// TwinCAT 3 PLC project PLC1
// ProgramVersion: 3.1.4024.0
// libraries:
//   Tc2_EtherCAT, * (Beckhoff Automation GmbH)
//   Tc2_MC2, * (Beckhoff Automation GmbH)
//   Tc2_Standard, * (Beckhoff Automation GmbH)
//   Tc2_System, * (Beckhoff Automation GmbH)
//   Tc3_Module, * (Beckhoff Automation GmbH)
// project tree:
//   DUTs/Dosing Pumps/ E_AccessType.TcDUT, E_DosingPump.TcDUT, E_ModbusDataType.TcDUT, ST_EmcoPumpModbusData.TcDUT, ST_ModbusRegister.TcDUT
//   DUTs/ E_ConveyorMoveType.TcDUT, E_DeviceState.TcDUT, E_LinActuatorMoveType.TcDUT, E_MoveState.TcDUT, E_TrayExchangeState.TcDUT, ST_INPUTS_LinAct.TcDUT, ST_INPUTS_POP.TcDUT, ST_INPUTS_LFT.TcDUT, ST_INPUTS_SequenceManager_POP.TcDUT, ST_INPUTS_StaticConv.TcDUT, ST_INPUTS_TrayCentre.TcDUT
//   DUTs/GVL/Inputs/Dosing Machine/Children/ ST_INPUTS_DosingMachine_Sump.TcDUT, ST_INPUTS_DosingMachine_Water.TcDUT
//   DUTs/GVL/Inputs/Dosing Machine/ ST_INPUTS_DosingMachine.TcDUT
//   DUTs/GVL/Inputs/RND_DM/Children/ ST_INPUTS_RND_DosingMachine_Sump.TcDUT, ST_INPUTS_RND_DosingMachine_Water.TcDUT
//   DUTs/GVL/Inputs/RND_DM/ ST_INPUTS_RND_DosingMachine.TcDUT
//   DUTs/GVL/Inputs/RND_SC/ ST_INPUTS_RND_LevelWaterControl.TcDUT, ST_INPUTS_RND_StackControl.TcDUT
//   DUTs/GVL/Inputs/RND_WTR/ ST_INPUTS_WaterTreatment_RND.TcDUT
//   DUTs/GVL/Inputs/Universal/ ST_INPUTS_BagFilters.TcDUT, ST_INPUTS_Calibration.TcDUT, ST_INPUTS_ControlLoop_BangBang.TcDUT, ST_INPUTS_ControlLoop_BangBangAnalog.TcDUT, ST_INPUTS_DosingPump.TcDUT, ST_INPUTS_Dosing_ControlLoop.TcDUT, ST_INPUTS_DrumFilter.TcDUT, ST_INPUTS_PumpDOL.TcDUT, ST_INPUTS_PumpVSD.TcDUT, ST_INPUTS_RND_HVAC_Indoor_Unit.TcDUT, ST_INPUTS_SequenceManager_DM.TcDUT, ST_INPUTS_SequenceManager_RND_DM.TcDUT, ST_INPUTS_Strainer.TcDUT, ST_INPUTS_Unit_OxyInjector.TcDUT, ST_INPUTS_Unit_OzoneGenerator.TcDUT, ST_INPUTS_Unit_RO_EDI.TcDUT, ST_INPUTS_Unit_UltraSonCleaner.TcDUT, ST_INPUTS_Unit_UVFilter.TcDUT, ST_INPUTS_ValveOnOFF.TcDUT
//   DUTs/GVL/Inputs/Water Treatment/ ST_INPUTS_WaterTreatment.TcDUT, ST_INPUTS_WaterTreatment_Water.TcDUT
//   DUTs/Machines/ E_MachineState.TcDUT, ST_DMComponents.TcDUT, ST_POPComponents.TcDUT, ST_LFTComponents.TcDUT, ST_RNDDMComponents.TcDUT, ST_RNDWTRComponents.TcDUT, ST_WTRComponents.TcDUT
//   DUTs/Universal/ E_AlarmPriority.TcDUT, E_DeviceMode.TcDUT, E_InterlockType.TcDUT, E_Job_Status.TcDUT, E_POP_Type.TcDUT, E_SensorType.TcDUT, E_SequenceList_DM.TcDUT, E_SequenceList_POP.TcDUT, E_SequenceList_RND_DM.TcDUT, E_SequenceList_WTR.TcDUT, E_SequenceState.TcDUT, ST_Alarm.TcDUT, ST_Crop.TcDUT, ST_CropJob.TcDUT, ST_HandShake_TrayMovement.TcDUT, ST_HVAC.TcDUT, ST_Interlock.TcDUT, ST_Modbus_ReadRequest.TcDUT, ST_Modbus_WriteRequest.TcDUT, ST_OEE.TcDUT, ST_PlantConfig.TcDUT, ST_SequenceStep.TcDUT, ST_Tray.TcDUT, ST_TrayExchangeHandshake.TcDUT, ST_Tray_1.TcDUT, ST_Tray_2.TcDUT
//   GVLs/ GVL.TcGVL, Inputs.TcGVL, IO_MAPPING.TcGVL, Safety.TcGVL
//   / MAIN.TcPOU, PlcTask.TcTTO
//   POUs/00 Interfaces/ FB_BaseDevice.TcPOU, FB_BaseMachine.TcPOU, FB_BaseMachine_1.TcPOU, FB_BaseSensor.TcPOU, FB_HandShake_TrayMovement.TcPOU, I_Device.TcIO, I_Machine.TcIO, I_PumpDosing.TcIO, I_PumpVSD.TcIO, I_Sensor.TcIO, I_Sequence.TcIO, I_ValveActuated.TcIO
//   POUs/01 Actuators/Dosing Machine/ FB_AutoClean_Filter_Bollfilter.TcPOU, FB_DosingPumpAgrowtek_R2.TcPOU, FB_DosingPumpAgrowtek_R2_1.TcPOU, FB_DosingPumpAgrowtek_R2_Batch.TcPOU, FB_DosingPumpPRISMA.TcPOU, FB_DrumFilter_Faivre120.TcPOU, FB_DrumFilter_Faivre60.TcPOU, FB_GasMonitoringPanel_CDA4022.TcPOU, FB_GasMonitoringPanel_CDA4022_R2.TcPOU, FB_HVAC_RND_Indoor_Unit.TcPOU, FB_HVAC_RND_ModbusApadtor.TcPOU, FB_LevelWaterControl.TcPOU, FB_OxygenInjector.TcPOU, FB_OxygenInjector_1.TcPOU, FB_OzoneGenerator.TcPOU, FB_PumpDOL_Onga413.TcPOU, FB_PumpDOL_Onga413_RND.TcPOU, FB_PumpVSD_DanfossFC202.TcPOU, FB_PumpVSD_GrundfosCUE.TcPOU, FB_UltraSonicCleaner.TcPOU, FB_Unit_RO_PW30_1.TcPOU, FB_Unit_RO_RND.TcPOU, FB_UVFilter_Pentair_EU40.TcPOU, FB_UVFilter_UltraAqua_MR4_220PP.TcPOU
//   POUs/01 Actuators/ FB_Valve_ONOFF_woMonitoring.TcPOU, FB_Valve_ONOFF_woMonitoring_1.TcPOU
//   POUs/01 Actuators/supersceded/ FB_DosingPumpAgrowtek.TcPOU
//   POUs/02 Sensors/Dosing Machine/ FB_Sensor_AtlasDO.TcPOU, FB_Sensor_AtlasEC.TcPOU, FB_Sensor_AtlasORP.TcPOU, FB_Sensor_AtlasPH.TcPOU, FB_Sensor_AtlasTEMP.TcPOU, FB_Sensor_GrowMedium_EC.TcPOU, FB_Sensor_GrowMedium_MOISTURE.TcPOU, FB_Sensor_GrowMedium_PH.TcPOU, FB_Sensor_IFM_PG2453.TcPOU, FB_Sensor_OceanControlsPressureTx_BVS006NA.TcPOU, FB_Sensor_SICKLevelSwitch_GRF18S.TcPOU
//   POUs/02 Sensors/ FB_DualRedundantSensor.TcPOU, FB_Sensor_4_20mA_Generic.TcPOU, FB_Sensor_VaisalaGMW90.TcPOU, FB_Sensor_VaisalaGMW90_R2.TcPOU, FB_Sensor_VaisalaGMW90_R2_1.TcPOU
//   POUs/03 Physical Entities/ FB_BagFilter.TcPOU, FB_Tank.TcPOU
//   POUs/04 Control Loops/Dosing Machine/ FB_BangBangControl.TcPOU, FB_BangBangControl_Analog.TcPOU, FB_BatchController_Dosing.TcPOU, FB_ControlLoop_DissOx.TcPOU, FB_ControlLoop_Dosing.TcPOU, FB_ControlLoop_HVAC.TcPOU, FB_ControlLoop_HVAC_1.TcPOU, FB_ControlLoop_MainPumpPressure.TcPOU, FB_ControlLoop_pH.TcPOU, FB_ControlLoop_PID.TcPOU, FB_ControlLoop_PID_HVAC.TcPOU, FB_ControlLoop_TankLevel.TcPOU
//   POUs/04 Control Loops/_ss/ FB_ControlLoop_Dosing_1.TcPOU
//   POUs/05 Sequences/Dosing Machine/ FB_SequenceDM_Calibrate.TcPOU, FB_SequenceDM_Drain.TcPOU, FB_SequenceDM_Fill.TcPOU, FB_SequenceDM_Main.TcPOU
//   POUs/05 Sequences/ FB_SequenceBase.TcPOU, FB_SequenceManager.TcPOU, FB_SequenceManager_1.TcPOU, FB_SequenceManager_ss.TcPOU
//   POUs/05 Sequences/POP/ FB_SequenceCONVEY_EXTEND.TcPOU, FB_SequenceCONVEY_RETRACT.TcPOU, FB_SequenceEXTEND_CONVEY.TcPOU, FB_SequenceGET_READY_EXTEND.TcPOU, FB_SequenceGET_READY_RETRACT.TcPOU, FB_SequenceRETRACT_CONVEY.TcPOU
//   POUs/05 Sequences/LFT/ FB_SequenceMOVE.TcPOU
//   POUs/05 Sequences/RnD Machines/ FB_SequenceRNDWTR_Main.TcPOU, FB_SequenceRND_Calibrate.TcPOU, FB_SequenceRND_Drain.TcPOU, FB_SequenceRND_Fill.TcPOU, FB_SequenceRND_FirstDose.TcPOU, FB_SequenceRND_Flush.TcPOU, FB_SequenceRND_Main.TcPOU
//   POUs/05 Sequences/Water Treatment/ FB_SequenceWTR_Calibrate.TcPOU, FB_SequenceWTR_Main.TcPOU
//   POUs/06 Machines/ FB_Machine_LFT.TcPOU
//   POUs/06 Machines/Others/ FB_Machine_DosingMachine.TcPOU, FB_Machine_RND_DosingMachine_R2.TcPOU, FB_Machine_RND_DosingMachine_R2_1.TcPOU, FB_Machine_WaterTreatment.TcPOU, FB_Machine_WaterTreatment_RND.TcPOU, FB_Stack_Controller.TcPOU, FB_Stack_Controller_RND.TcPOU
//   POUs/06 Machines/_ss/ FB_Machine_DosingMachine_TEST2.TcPOU, FB_Machine_RND_DosingMachine.TcPOU
//   POUs/07 Systems/RND/ FB_System_RND_GasMonitoring.TcPOU, FB_System_RND_GasMonitoring_R2.TcPOU, FB_System_RND_HVAC.TcPOU
//   POUs/97 Signal Conditioning/ FB_SigCond_MovingAverage.TcPOU
//   POUs/99 Utilities/ FB_HealthMonitoring.TcPOU, FB_InterlockManager.TcPOU, FB_ModbusManager.TcPOU, FB_ModbusMaster_R2.TcPOU, FB_RS485_CardRead.TcPOU, FB_RS485_CardWrite.TcPOU, FB_SensorVirtual_Vaisala.TcPOU, FB_TimeStampProvider.TcPOU
//   POUs/99 Utilities/_ss/ FB_ModbusManager_1.TcPOU, FB_ModbusMaster.TcPOU, FB_ModbusMaster_R2_1.TcPOU
//   POUs/LFT/ E_AxisNumberCoE.TcDUT, E_CoEService.TcDUT, E_ConfigurationStateCoE.TcDUT, E_MovidriveB_OpMode.TcDUT, FB_AutoGreaser.TcPOU, FB_Lift.TcPOU, FB_LiftArm.TcPOU, FB_ParameterCoE_ReadWrite_GenC.TcPOU, FB_SEW_MovidriveB.TcPOU, ST_StackDestination.TcDUT
//   POUs/POP/ FB_ActuatorLinear.TcPOU, FB_AutoSwitch.TcPOU, FB_BaseMotor.TcPOU, FB_LinearActuator_Elec.TcPOU, FB_LinearActuator_Pneumatic.TcPOU, FB_Sensor_OMRON_E3AS.TcPOU, FB_StaticConveyor.TcPOU
// real-time tasks:
//   TASK PlcTask: cycle T#10ms, priority 20, ADS port 350
// I/O:
//   DEVICE CONTROL_BOX, AmsNetId 192.168.1.31.2.1
//     Term 1 (EK1200) [EK1200-5000 EtherCAT Power supply (2A E-Bus)]
//       Term 8 (EL6070) [EL6070 1Ch. Licensing-Terminal]
//       Term 9 (EL6910) [EL6910, TwinSAFE PLC]
//       Term 10 (EL1904) [EL1904, 4 Ch. Safety Input 24V, TwinSAFE]
//         modules: Module 1 (FSOES)
//       Term 11 (EL1008) [EL1008 8Ch. Dig. Input 24V, 3ms]
//       Term 12 (EL1904) [EL1904, 4 Ch. Safety Input 24V, TwinSAFE]
//         modules: Module 1 (FSOES)
//       Term 13 (EL1904) [EL1904, 4 Ch. Safety Input 24V, TwinSAFE]
//         modules: Module 1 (FSOES)
//       Term 14 (EL2008) [EL2008 8Ch. Dig. Output 24V, 0.5A]
//       Term 15 (EL2904) [EL2904, 4 Ch. Safety Output 24V, 0.5A, TwinSAFE]
//         modules: Module 1 (FSOES), Module 2 (DO)
//       Term 10 (EL9011) [EL9011 End Terminal]
//   DEVICE Device 4 (EtherCAT), AmsNetId 192.168.1.31.5.1
//     Box 1 (EP1008-0002) [EP1008-0002 8 Ch. Dig. Input 24V, 3ms, M12]
//     Box 2 (EP2308-0002) [EP2308-0002 4 CH. Dig. In, 3ms, 4 Ch. Dig. Out 24V, 0,5A, M12]
//     Drive 3 (MOVIDRIVE+DFE24) [MOVIDRIVE+DFE24]
// variable links:
//   CONTROL_BOX <-> CONTROL_BOX/Term 1 (EK1200)/Term 12 (EL1904)
//     Term 1 (EK1200)/Term 9 (EL6910)/ConnectionOutputs/Message_3 RxPDO <-> Module 1 (FSOES)/TxPDO/FSOE
//   CONTROL_BOX <-> CONTROL_BOX/Term 1 (EK1200)/Term 9 (EL6910)
//     Term 1 (EK1200)/Term 10 (EL1904)/Module 1 (FSOES)/RxPDO/FSOE <-> ConnectionInputs/Message_2 TxPDO
//     Term 1 (EK1200)/Term 12 (EL1904)/Module 1 (FSOES)/RxPDO/FSOE <-> ConnectionInputs/Message_3 TxPDO
//     Term 1 (EK1200)/Term 13 (EL1904)/Module 1 (FSOES)/RxPDO/FSOE <-> ConnectionInputs/Message_4 TxPDO
//     Term 1 (EK1200)/Term 15 (EL2904)/Module 1 (FSOES)/RxPDO/FSOE <-> ConnectionInputs/Message_5 TxPDO
//     Term 1 (EK1200)/Term 10 (EL1904)/Module 1 (FSOES)/TxPDO/FSOE <-> ConnectionOutputs/Message_2 RxPDO
//     Term 1 (EK1200)/Term 13 (EL1904)/Module 1 (FSOES)/TxPDO/FSOE <-> ConnectionOutputs/Message_4 RxPDO
//     Term 1 (EK1200)/Term 15 (EL2904)/Module 1 (FSOES)/TxPDO/FSOE <-> ConnectionOutputs/Message_5 RxPDO
//   PLC1/PLC1 Instance <-> CONTROL_BOX/Term 1 (EK1200)/Term 11 (EL1008)
//     PlcTask Inputs/MAIN.fbMachine_Lift.fbSensor_PressSwitch.bRawInput <-> Channel 3/Input
//   PLC1/PLC1 Instance <-> CONTROL_BOX/Term 1 (EK1200)/Term 14 (EL2008)
//     PlcTask Outputs/MAIN.fbMachine_Lift.bLOCK_CTRL <-> Channel 3/Output
//     PlcTask Outputs/MAIN.fbMachine_Lift.bPWR_CTRL <-> Channel 1/Output
//   PLC1/PLC1 Instance <-> CONTROL_BOX/Term 1 (EK1200)/Term 9 (EL6910)
//     PlcTask Outputs/Safety.bSafetyErrorAcknowledge <-> StandardOutputs/Standard In Var 1
//     PlcTask Outputs/Safety.bSafety_Run_Stop <-> StandardOutputs/Standard In Var 7
//   PLC1/PLC1 Instance <-> Device 4 (EtherCAT)/Box 1 (EP1008-0002)
//     PlcTask Inputs/MAIN.fbMachine_Lift.fbSensor_LiftBrake_Left.bRawInput <-> Channel 8/Input
//     PlcTask Inputs/MAIN.fbMachine_Lift.fbSensor_LiftBrake_Right.bRawInput <-> Channel 7/Input
//     PlcTask Inputs/MAIN.fbMachine_Lift.fbSensor_Lift_Bottom.bRawInput <-> Channel 3/Input
//     PlcTask Inputs/MAIN.fbMachine_Lift.fbSensor_Lift_Home.bRawInput <-> Channel 1/Input
//     PlcTask Inputs/MAIN.fbMachine_Lift.fbSensor_Lift_Top.bRawInput <-> Channel 2/Input
//   PLC1/PLC1 Instance <-> Device 4 (EtherCAT)/Box 2 (EP2308-0002)
//     PlcTask Outputs/MAIN.bGreaser <-> Channel 5/Output
//     PlcTask Outputs/MAIN.bGreaser2 <-> Channel 6/Output
//     PlcTask Outputs/MAIN.fbMachine_Lift.fbValve_Brake.bValveOutput <-> Channel 8/Output
//     PlcTask Outputs/MAIN.fbMachine_Lift.fbValve_Vacuum.bValveOutput <-> Channel 7/Output

CONFIGURATION PLC1
    RESOURCE PLC ON TwinCAT3
        TASK PlcTask(INTERVAL := T#10ms, PRIORITY := 20);
        PROGRAM MAIN WITH PlcTask : MAIN;
    END_RESOURCE
END_CONFIGURATION

// ---- DUTs/Dosing Pumps/E_AccessType.TcDUT
{attribute 'qualified_only'}
{attribute 'strict'}
TYPE E_AccessType :
(
	READ,
	WRITE,
	READWRITE
);
END_TYPE

// ---- DUTs/Dosing Pumps/E_DosingPump.TcDUT
{attribute 'qualified_only'}
{attribute 'strict'}
TYPE E_DosingPump :
(
	PH_UP := 0,
	PH_DOWN := 1,
	NUTRIENT_A := 2,
	NUTRIENT_B := 3,
	NUTRIENT_C := 4
);
END_TYPE

// ---- DUTs/Dosing Pumps/E_ModbusDataType.TcDUT
{attribute 'qualified_only'}
{attribute 'strict'}
TYPE E_ModbusDataType :
(
	uint16,
	uint32,
	uint64
);
END_TYPE

// ---- DUTs/Dosing Pumps/ST_EmcoPumpModbusData.TcDUT
TYPE ST_EmcoPumpModbusData :
STRUCT
	ALARM_Level_Alarm:  UINT;
	ALARM_Pump_Status_When_Level_Alarm_Occurs:  UINT;
	ALARM_Stand_By:  UINT;
	ALARM_Overflow:  UINT;
	ALARM_Temperature:  UINT;
	ALARM_No_Input:  UINT;
	ALARM_Overpressure:  UINT;
	DOSAGE_Dosage_Schedule:  UDINT;
	DOSAGE_Frequency:  UDINT;
	SETTINGS_Level_Alarm:  UINT;
	SETTINGS_Level_Alarm_Contact:  UINT;
	SETTINGS_Reserve_Level_Alarm:  UDINT;
	SETTINGS_Unit:  UINT;
	MODE_Working_Mode:  UINT;
	SETTINGS_Water_Meter_Input_Unit_Of_Measure:  UINT;
	SETTINGS_Water_Meter_Input_Value:  UINT;
	STATISTICS_Partial_Statistics_Dosato:  ULINT;
	STATISTICS_Partial_Statistics_Counter:  ULINT;
	STATISTICS_Partial_Statistics_Dosato_In_The_Last_24H:  ULINT;
	STATISTICS_Partial_Statistics_Counter_In_The_Last_24H:  ULINT;
	STATISTICS_Partial_Statistics_Reset_The_Last_Time_Hrs:  UINT;
	STATISTICS_Partial_Statistics_Reset_The_Last_Time_Mins:  UINT;
	STATISTICS_Partial_Statistics_Reset_The_Last_Time_Seconds:  UINT;
	STATISTICS_Partial_Statistics_Date_Last_Reset_Day:  UINT;
	STATISTICS_Partial_Statistics_Date_Last_Reset_Month:  UINT;
	STATISTICS_Partial_Statistics_Date_Last_Reset_Year:  UINT;
	STATISTICS_Statistics_Total_Total_Dosage:  ULINT;
	STATISTICS_Statistics_Total_Counter:  ULINT;
	MODE_ON_OFF:  UINT;
	SETTINGS_Timeout_Val:  UINT;
	SETTINGS_Overflow_Val:  UINT;
	SETTINGS_Delay:  UINT;
	MODE_Constant_Mode:  UDINT;
	MODE_Mode_Ppm:  UDINT;
	MODE_Mode_Ppm_Concentration:  UINT;
	MODE_Mode_Perc:  UDINT;
	MODE_Mode_Perc_Concentration:  UINT;
	MODE_Mode_Mlq:  UDINT;
	MODE_Mode_Mlq_Concentration:  UINT;
	MODE_Method_Volt_Volt_High_Value:  UINT;
	MODE_Method_Volt_Volt_Low_Value:  UINT;
	MODE_Method_Volt_High_Dose:  UDINT;
	MODE_Mode_Volt_Low_Dose:  UDINT;
	MODE_Method_Ma_Ma_High_Value:  UINT;
	MODE_Method_Ma_Ma_Low_Value:  UINT;
	MODE_Method_Ma_High_Dosage:  UDINT;
	MODE_Method_Ma_Low_Dosage:  UDINT;
	MODE_Pulse_Mode_Pulse_High_Value:  UINT;
	MODE_Pulse_Mode_Pulse_Low_Value:  UINT;
	MODE_Pulse_Mode_High_Dose:  UDINT;
	MODE_Pulse_Low_Dose:  UDINT;
	MODE_Method_Pause_Minutes_Work_Work:  UINT;
	MODE_Method_Pause_Minutes_Of_Work_Pause:  UINT;
	MODE_Method_Pause_Quantity_Work_To_Dose:  UDINT;
	SETTINGS_Flow:  UDINT;
	SETTINGS_Slow_Mode:  UINT;
	SETTINGS_Alarm_Output:  UINT;
	SETTINGS_Alarm_Output_Contact_0_No_1_Nc:  UINT;
	SETTINGS_Alarm_Output_Alert_Level:  UINT;
	SETTINGS_Alarm_Out_Standby:  UINT;
	SETTINGS_Alarm_Output_Alarm_Overflow:  UINT;
	SETTINGS_Exit_Alarm_Temperature_Alarm:  UINT;
	SETTINGS_Alarm_Output_No_Alarm_Input:  UINT;
	SETTINGS_Alarm_Output_For_Overpressure:  UINT;
	SETTINGS_Standby:  UINT;
	SETTINGS_Standby_Contact_No_0_1_Nc:  UINT;
	SETTINGS_Constant_Dosage_With_External_Input_Enable:  UINT;
	SETTINGS_Constant_Dosage_With_External_Input_No_0_1_Nc:  UINT;
	SETTINGS_Constant_Dosage_With_External_Input_Dosing_Speed:  UDINT;
	MODE_Cc_Pulse_Mode:  UDINT;
	MODE_Batch_Mode_External_Quantity:  UDINT;
	MODE_Batch_Mode_External_Contact_1_Nc_0_No:  UINT;

END_STRUCT
END_TYPE

// ---- DUTs/Dosing Pumps/ST_ModbusRegister.TcDUT
TYPE ST_ModbusRegister :
STRUCT
	Reg_Adress: UDINT;
	Num_Bytes: INT;
	Value_Type: E_ModbusDataType;
	Description: STRING;
	AccessType: E_AccessType;
	Value: ARRAY[1..4] OF WORD;
END_STRUCT
END_TYPE

// ---- DUTs/E_ConveyorMoveType.TcDUT
{attribute 'qualified_only'}
{attribute 'strict'}
TYPE E_ConveyorMoveType :
(
	FORWARD,
	FORWARD_SLOW,
	REVERSE,
	REVERSE_SLOW,
	STOP
);
END_TYPE

// ---- DUTs/E_DeviceState.TcDUT
{attribute 'qualified_only'}
{attribute 'strict'}
TYPE E_DeviceState :
(
	// Motors & Pumps
	IDLE,
	STARTING,
	RUNNING ,
	REVERSE ,
	STOPPING,
	
	// Universal
	FAULTED ,
	ENABLED  ,
	
	// Tanks & Sumps
	// Sensors 
	HIGH_HIGH,
	HIGH ,
	LOW ,
	LOW_LOW,
	
	// Sensors 
	IN_RANGE ,
	OUT_OF_RANGE,
	
	
	// Valves
	OPEN ,
	OPENING,
	CLOSED ,
	CLOSING,
	
	// Other ON/OFF devices (e.g. oxygen injector, UV filter)
	TURNING_ON,
	ON ,
	TURNING_OFF,
	OFF,
	
	// Sensors
	CAL_STEP1,
	CAL_STEP2,
	CAL_STEP3,
	CAL_STEP4,
	
	// Linear Actuator
	EXTENDING,
	EXTENDED,
	RETRACTING,
	RETRACTED
	
);
END_TYPE

// ---- DUTs/E_LinActuatorMoveType.TcDUT
{attribute 'qualified_only'}
{attribute 'strict'}
TYPE E_LinActuatorMoveType :
(
	EXTEND,
	EXTEND_SLOW,
	RETRACT,
	RETRACT_SLOW,
	STOP
);
END_TYPE

// ---- DUTs/E_MoveState.TcDUT
TYPE E_MoveState :
(
	MOVESTATE_INIT,
	MOVESTATE_ENABLE,
	MOVESTATE_FORWARD,
	MOVESTATE_BACKWARDS,
	MOVESTATE_BACKWARDSSLOW,
	MOVESTATE_NEWTARGETPOSITION,
	MOVESTATE_ERROR,
	MOVESTATE_RESET
) UDINT;
END_TYPE

// ---- DUTs/E_TrayExchangeState.TcDUT
{attribute 'qualified_only'}
{attribute 'strict'}
TYPE E_TrayExchangeState :
(
	IDLE,
	REQUESTED,
	ACCEPTED,
	IN_PROGRESS,
	COMPLETED
);
END_TYPE

// ---- DUTs/GVL/Inputs/Dosing Machine/Children/ST_INPUTS_DosingMachine_Sump.TcDUT
TYPE ST_INPUTS_DosingMachine_Sump :
STRUCT

	Level_LOW_LOW_Limit:    	UINT;
	Level_LOW_Limit:    		UINT;
	Level_HIGH_Limit:    	UINT;
	Level_HIGH_HIGH_Limit:   UINT;
	Level_Setpoint:    		UINT;
	
	Pressure_Dosing_LOW_Limit:    	UINT;
	Pressure_Dosing_HIGH_Limit:    	UINT;
		


END_STRUCT
END_TYPE

// ---- DUTs/GVL/Inputs/Dosing Machine/Children/ST_INPUTS_DosingMachine_Water.TcDUT
TYPE ST_INPUTS_DosingMachine_Water :
STRUCT
	EC_Alarm_HIGH:	REAL;
	EC_Alarm_LOW:	REAL;
	EC_LOW_Limit:    UINT; // short
	EC_HIGH_Limit:    UINT; // float
	EC_SetPoint:    UINT; // double
	EC_Selection:    UINT;
	
	PH_Alarm_HIGH:	REAL;
	PH_Alarm_LOW:	REAL;
	PH_LOW_Limit:    REAL;
	PH_HIGH_Limit:    REAL;
	PH_SetPoint:    REAL;
	PH_Selection:    REAL;
	
	DO_Alarm_HIGH:	REAL;
	DO_Alarm_LOW:	REAL;
	DO_LOW_Limit:    REAL;
	DO_HIGH_Limit:    REAL;
	DO_SetPoint:    REAL;
	DO_Selection:    REAL;
	
	ORP_Alarm_HIGH:	REAL;
	ORP_Alarm_LOW:	REAL;
	ORP_LOW_Limit:    REAL;
	ORP_HIGH_Limit:    REAL;
	ORP_SetPoint:    REAL;
	ORP_Selection:    REAL;
	
	Temp_Alarm_HIGH:	REAL;
	Temp_Alarm_LOW:	REAL;
	Temp_LOW_Limit:    REAL;
	Temp_HIGH_Limit:    REAL;
	Temp_SetPoint:    REAL;
	Temp_Selection:    REAL;
	
	Calibrate_PH: BOOL;
	Calibrate_EC: BOOL;
	Calibrate_DO: BOOL;
	Calibrate_ORP: BOOL;
	Calibrate_TEMP: BOOL;


END_STRUCT
END_TYPE

// ---- DUTs/GVL/Inputs/Dosing Machine/ST_INPUTS_DosingMachine.TcDUT
TYPE ST_INPUTS_DosingMachine:
STRUCT

	Pump_MainPumpSelection_A_1_B_0: UINT;
	

	stWaterQuality: ST_INPUTS_DosingMachine_Water;
	stSumpDosing: ST_INPUTS_DosingMachine_Sump;
	
	stSequenceManager: 			ST_INPUTS_SequenceManager_DM;
	stValve_DosingSupply: ST_INPUTS_ValveOnOFF;
	stValve_IrrigatorSupply: ST_INPUTS_ValveOnOFF;
	stValve_WasteWaterReturn: ST_INPUTS_ValveOnOFF;
	stUnit_OxyInjector: ST_INPUTS_Unit_OxyInjector;
	stUnit_UltraSonCleaner: ST_INPUTS_Unit_UltraSonCleaner;
	stStrainer: ST_INPUTS_Strainer;
	stUVFilter: ST_INPUTS_Unit_UVFilter;
	stDosingPump_phUp: ST_INPUTS_DosingPump;
	stDosingPump_phDown: ST_INPUTS_DosingPump;	
	stDosingPump_NutrientA: ST_INPUTS_DosingPump;	
	stDosingPump_NutrientB: ST_INPUTS_DosingPump;	
	stDosingPump_NutrientC: ST_INPUTS_DosingPump;	
	stPump_MainPumpA: ST_INPUTS_PumpVSD;
	stPump_MainPumpB: ST_INPUTS_PumpVSD;
	stControlLoopDosing_Nutrient: ST_INPUTS_Dosing_ControlLoop;
	stControlLoopDosing_PH: ST_INPUTS_Dosing_ControlLoop;
	


END_STRUCT
END_TYPE

// ---- DUTs/GVL/Inputs/RND_DM/Children/ST_INPUTS_RND_DosingMachine_Sump.TcDUT
TYPE ST_INPUTS_RND_DosingMachine_Sump :
STRUCT

	Level_LOW_LOW_Limit:    	UINT;
	Level_LOW_Limit:    		UINT;
	Level_HIGH_Limit:    	UINT;
	Level_HIGH_HIGH_Limit:   UINT;
	Level_Setpoint:    		UINT;
	
	Pressure_Dosing_LOW_Limit:    	UINT;
	Pressure_Dosing_HIGH_Limit:    	UINT;
		


END_STRUCT
END_TYPE

// ---- DUTs/GVL/Inputs/RND_DM/Children/ST_INPUTS_RND_DosingMachine_Water.TcDUT
TYPE ST_INPUTS_RND_DosingMachine_Water :
STRUCT
	EC_LOW_Limit:    REAL; // short
	EC_HIGH_Limit:    REAL; // float
	EC_LOW_Alarm:    REAL; // short
	EC_HIGH_Alarm:    REAL; // float
	EC_SetPoint:    REAL; // double
	EC_Selection:    REAL;
	
	EC_Enforce_Low: BOOL;  // if this is true then irrigation will be inhibited
	EC_Enforce_High: BOOL;  // if this is true then irrigation will be inhibited
	
	PH_LOW_Limit:    REAL;
	PH_HIGH_Limit:    REAL;
	PH_LOW_Alarm:    REAL;
	PH_HIGH_Alarm:    REAL;
	PH_SetPoint:    REAL;
	PH_Selection:    REAL;
	
	PH_Enforce_Low: BOOL;  // if this is true then irrigation will be inhibited
	PH_Enforce_High: BOOL;  // if this is true then irrigation will be inhibited
	
	DO_LOW_Limit:    REAL;
	DO_HIGH_Limit:    REAL;
	DO_LOW_Alarm:    REAL;
	DO_HIGH_Alarm:    REAL;
	DO_SetPoint:    REAL;
	DO_Selection:    REAL;
	
	DO_Enforce_Low: BOOL;  // if this is true then irrigation will be inhibited
	DO_Enforce_High: BOOL;  // if this is true then irrigation will be inhibited
	
	ORP_LOW_Limit:    REAL;
	ORP_HIGH_Limit:    REAL;
	ORP_LOW_Alarm:    REAL;
	ORP_HIGH_Alarm:    REAL;
	ORP_SetPoint:    REAL;
	ORP_Selection:    REAL;
	
	ORP_Enforce_Low: BOOL;  // if this is true then irrigation will be inhibited
	ORP_Enforce_High: BOOL;  // if this is true then irrigation will be inhibited
	
	Temp_LOW_Limit:    REAL;
	Temp_HIGH_Limit:    REAL;
	Temp_LOW_Alarm:    REAL;
	Temp_HIGH_Alarm:    REAL;
	Temp_SetPoint:    REAL;
	Temp_Selection:    REAL;
	
	Temp_Enforce_Low: BOOL;  // if this is true then irrigation will be inhibited
	Temp_Enforce_High: BOOL;  // if this is true then irrigation will be inhibited
	
	Calibrate_PH: BOOL;
	Calibrate_EC: BOOL;
	Calibrate_DO: BOOL;
	Calibrate_ORP: BOOL;
	Calibrate_TEMP: BOOL;


END_STRUCT
END_TYPE

// ---- DUTs/GVL/Inputs/RND_DM/ST_INPUTS_RND_DosingMachine.TcDUT
TYPE ST_INPUTS_RND_DosingMachine:
STRUCT

	stWaterQuality: 				ST_INPUTS_RND_DosingMachine_Water;
	stSumpDosing: 					ST_INPUTS_RND_DosingMachine_Sump;
	stSequenceManager: 				ST_INPUTS_SequenceManager_RND_DM;
	stValve_ROSupply: 				ST_INPUTS_ValveOnOFF;
	stValve_IrrigatorSupply: 		ST_INPUTS_ValveOnOFF;
	stUVFilter: 					ST_INPUTS_Unit_UVFilter; // this is the same as the main dosing machine uv filter - are there differences?
	stDosingPump_phUp: 				ST_INPUTS_DosingPump;
	stDosingPump_phDown: 			ST_INPUTS_DosingPump;	
	stDosingPump_NutrientA: 		ST_INPUTS_DosingPump;	
	stDosingPump_NutrientB: 		ST_INPUTS_DosingPump;	
	stDosingPump_NutrientC: 		ST_INPUTS_DosingPump;	
	stPump_MainPumpA: 				ST_INPUTS_PumpDOL;
	stControlLoopDosing_Nutrient: 	ST_INPUTS_Dosing_ControlLoop;
	stControlLoopDosing_PH: 		ST_INPUTS_Dosing_ControlLoop;
	stCalibration:					ST_INPUTS_Calibration;

	
	bParamsInitialised: BOOL := FALSE;
	
	// stValve_WasteWaterReturn: ST_INPUTS_ValveOnOFF; <-- should be there a waste water return?
	// stUnit_OxyInjector: ST_INPUTS_Unit_OxyInjector;  // this is passive in the R&D rooms
	// stUnit_UltraSonCleaner: ST_INPUTS_Unit_UltraSonCleaner; // not included in R&D system
	// stDrumFilter: ST_INPUTS_DrumFilter; // not included in R&D system

END_STRUCT
END_TYPE

// ---- DUTs/GVL/Inputs/RND_SC/ST_INPUTS_RND_LevelWaterControl.TcDUT
TYPE ST_INPUTS_RND_LevelWaterControl :
STRUCT
	
	Valve: 	ST_INPUTS_ValveOnOFF;
	MinutesOff : INT;
	MinutesOn : INT;
	
	//TimeUntilOn: INT; // number of seconds until the irrigator is turned on (0s of the irrigator is on)

END_STRUCT
END_TYPE

// ---- DUTs/GVL/Inputs/RND_SC/ST_INPUTS_RND_StackControl.TcDUT
TYPE ST_INPUTS_RND_StackControl :
STRUCT
	

	HumidityControl: 					ST_INPUTS_ControlLoop_BangBang;
	CO2Control: 						ST_INPUTS_ControlLoop_BangBang;
	TemperatureControl:					ST_INPUTS_ControlLoop_BangBangAnalog;
	
	FanControl_Exhaust:					ST_INPUTS_ControlLoop_BangBang;
	FanControl_Circulation:				ST_INPUTS_ControlLoop_BangBang;
	
	LevelWaterControls:	ARRAY[0..1] OF  ST_INPUTS_RND_LevelWaterControl;
	
	bParamsInitialised: BOOL := FALSE;
	
	bWaterQualityGood: BOOL := FALSE; // The dosing machine writes to this to inhibit irrigator action in the Stack Controller
	
	//bIrrigatorValve_NC_1_NO_0: BOOL := FALSE;
	
	// bIrrigValve_NC_1_NO_0: BOOL := FALSE;
	
END_STRUCT
END_TYPE

// ---- DUTs/GVL/Inputs/RND_WTR/ST_INPUTS_WaterTreatment_RND.TcDUT
TYPE ST_INPUTS_WaterTreatment_RND :
STRUCT
	
	//stSequenceManager: ST_INPUTS_SequenceManager_DM;
	//stPump_CleanWaterPumpA: ST_INPUTS_PumpVSD;
	stUnit_RO_EDI: ST_INPUTS_Unit_RO_EDI;
	//stValve_DM1_Supply: ST_INPUTS_ValveOnOFF;
	
	stSequenceManager: 	ST_INPUTS_SequenceManager_RND_DM;

END_STRUCT
END_TYPE

// ---- DUTs/GVL/Inputs/Universal/ST_INPUTS_BagFilters.TcDUT
TYPE ST_INPUTS_BagFilters:
STRUCT
	
	Filter1_MaxDiffPressure:    UINT;
	Filter2_MaxDiffPressure:    UINT;

END_STRUCT
END_TYPE

// ---- DUTs/GVL/Inputs/Universal/ST_INPUTS_Calibration.TcDUT
TYPE ST_INPUTS_Calibration :
STRUCT
	Start_DO: BOOL;
	Step1_DO: BOOL;
	Step2_DO: BOOL;
	Complete_DO: BOOL;
	
	Start_EC: BOOL;
	Step1_EC: BOOL;
	Step2_EC: BOOL;
	Complete_EC: BOOL;

	Start_PH: BOOL;
	Step1_PH: BOOL;
	Step2_PH: BOOL;
	Step3_PH: BOOL;
	Complete_PH: BOOL;
	
	Start_ORP: BOOL;
	Step1_ORP: BOOL;
	Complete_ORP: BOOL;
	
	Start_TMP: BOOL;
	Step1_TMP: BOOL;
	Complete_TMP: BOOL;
	
	Cal_SoilSensor_EC1: BOOL;
	Cal_SoilSensor_EC2: BOOL;
	Cal_SoilSensor_PH1: BOOL;
	Cal_SoilSensor_PH2: BOOL;
	Cal_SoilSensor_Moisture1: BOOL;
	Cal_SoilSensor_Moisture2: BOOL;
	
END_STRUCT
END_TYPE

// ---- DUTs/GVL/Inputs/Universal/ST_INPUTS_ControlLoop_BangBang.TcDUT
TYPE ST_INPUTS_ControlLoop_BangBang :
STRUCT
	
	rAlarmHigh : 			REAL;
	rAlarmLow : 			REAL;
	rLimitHigh : 			REAL; // the upper limit of the desirable range (when the downward adjustment is activated)
	rLimitLow : 			REAL; // lower limit of the desirable range (when the upward adjustment is activated)
	nAdjustDelay : 			REAL; // min time in seconds between adjustments
	nAdjustDownDuration : 	REAL; // time in seconds that the downward adjustment output is turned on when performing a downward adjustment
	nAdjustUpDuration : 	REAL; // time in seconds that the upward adjustment output is turned on when performing a upward adjustment
	bEnabled : 				BOOL; 
	Mode:     				E_CTRL_MODE;

END_STRUCT
END_TYPE

// ---- DUTs/GVL/Inputs/Universal/ST_INPUTS_ControlLoop_BangBangAnalog.TcDUT
TYPE ST_INPUTS_ControlLoop_BangBangAnalog :
STRUCT

	rAlarmHigh : REAL;
	rAlarmLow : REAL;
	rLimitHigh : REAL; // the upper limit of the desirable range (when the downward adjustment is activated)
	rLimitLow : REAL; // lower limit of the desirable range (when the upward adjustment is activated)
	nAdjustDelay : INT; // min time in seconds between adjustments
	nAdjustDownIncrement : REAL; // amount to adjust control value if the actual value is above setpoint 
	nAdjustUpIncrement : REAL; // amount to adjust control value if the actual value is below setpoint
	bEnabled : BOOL; 
	Mode:   E_CTRL_MODE;	
	
	rDegPerHr: REAL;
	
END_STRUCT
END_TYPE

// ---- DUTs/GVL/Inputs/Universal/ST_INPUTS_DosingPump.TcDUT
TYPE ST_INPUTS_DosingPump :
STRUCT
	
	Mode:     E_DeviceMode;
	Command:     E_DeviceState;
	DoseQty_mls:     UINT;
	DoseRate_mlph:     UINT;
	ModbusSlaveID:     UINT;
	ResetPumpStatistics:     BOOL;
	Dose_OneShot: 		BOOL;
	
	InitialDose: BOOL; // this is a placeholder for when we bring in the new dosing pump fb for initial dose
	

END_STRUCT
END_TYPE

// ---- DUTs/GVL/Inputs/Universal/ST_INPUTS_Dosing_ControlLoop.TcDUT
TYPE ST_INPUTS_Dosing_ControlLoop :
STRUCT
	
	Setpoint:     	REAL;
	SetpointBand:   REAL;
	ManSyncVal:     REAL;
	Sync:     		BOOL;
	Hold:     		BOOL;
	Mode:     		E_CTRL_MODE;
	ARWactive:     	BOOL;
	
	CtrlCycleTime:  UINT;
	TaskCycleTime:  UINT;
	Kp:     		REAL;
	Tn:     		UINT;
	Tv:     		UINT;
	Td:     		UINT;
	OutMaxLimit:    REAL;
	OutMinLimit:    REAL;
	PInTheFeedbackPath:     BOOL;
	DInTheFeedbackPath:     BOOL;
	ARWOnIPartOnly:     	BOOL;
	
	MaxDoseRate:   		UINT;
	MinDoseRate:    	UINT;
	TimeBetweenDoses:   UINT;


END_STRUCT
END_TYPE

// ---- DUTs/GVL/Inputs/Universal/ST_INPUTS_DrumFilter.TcDUT
TYPE ST_INPUTS_DrumFilter:
STRUCT
	
	Mode:     		E_DeviceMode;
	Command:     E_DeviceState;

END_STRUCT
END_TYPE

// ---- DUTs/GVL/Inputs/Universal/ST_INPUTS_PumpDOL.TcDUT
TYPE ST_INPUTS_PumpDOL:
STRUCT
	
	Mode:     		E_DeviceMode;
	Command:     E_DeviceState;

END_STRUCT
END_TYPE

// ---- DUTs/GVL/Inputs/Universal/ST_INPUTS_PumpVSD.TcDUT
TYPE ST_INPUTS_PumpVSD:
STRUCT
	
	
	Mode:     			E_DeviceMode;
	Command:     		E_DeviceState;
	MinFrequency:     	UINT;
	CommandFrequency:   UINT;
	
	


END_STRUCT
END_TYPE

// ---- DUTs/GVL/Inputs/Universal/ST_INPUTS_RND_HVAC_Indoor_Unit.TcDUT
TYPE ST_INPUTS_RND_HVAC_Indoor_Unit :
STRUCT
	
	On_Off_1_0:		BOOL;
	TempSetPoint:	REAL;
	
END_STRUCT
END_TYPE

// ---- DUTs/GVL/Inputs/Universal/ST_INPUTS_SequenceManager_DM.TcDUT
TYPE ST_INPUTS_SequenceManager_DM:
STRUCT
	
	Sequence_Selected: E_SequenceList_DM;
	Sequence_Command: E_SequenceState;
	Sequence_Ack_Interlock: BOOL;
	
	
END_STRUCT
END_TYPE

// ---- DUTs/GVL/Inputs/Universal/ST_INPUTS_SequenceManager_RND_DM.TcDUT
TYPE ST_INPUTS_SequenceManager_RND_DM:
STRUCT
	
	Sequence_Previous: E_SequenceList_RND_DM; // used for resuming previous sequence after calibrartion
	Sequence_Selected: E_SequenceList_RND_DM;
	Sequence_Command: E_SequenceState;
	Sequence_Ack_Interlock: BOOL;
	
	
END_STRUCT
END_TYPE

// ---- DUTs/GVL/Inputs/Universal/ST_INPUTS_Strainer.TcDUT
TYPE ST_INPUTS_Strainer:
STRUCT
	
	Mode:     	E_DeviceMode;
	Command:     E_DeviceState;

END_STRUCT
END_TYPE

// ---- DUTs/GVL/Inputs/Universal/ST_INPUTS_Unit_OxyInjector.TcDUT
TYPE ST_INPUTS_Unit_OxyInjector:
STRUCT
	
	Mode:     	 E_DeviceMode;
	Command:     E_DeviceState;

END_STRUCT
END_TYPE

// ---- DUTs/GVL/Inputs/Universal/ST_INPUTS_Unit_OzoneGenerator.TcDUT
TYPE ST_INPUTS_Unit_OzoneGenerator:
STRUCT
	
	Mode:     		E_DeviceMode;
	Command:     E_DeviceState;

END_STRUCT
END_TYPE

// ---- DUTs/GVL/Inputs/Universal/ST_INPUTS_Unit_RO_EDI.TcDUT
TYPE ST_INPUTS_Unit_RO_EDI:
STRUCT
	
	Mode:     		E_DeviceMode;
	Command:     	E_DeviceState;

END_STRUCT
END_TYPE

// ---- DUTs/GVL/Inputs/Universal/ST_INPUTS_Unit_UltraSonCleaner.TcDUT
TYPE ST_INPUTS_Unit_UltraSonCleaner:
STRUCT
	
	Mode:     		E_DeviceMode;
	Command:     E_DeviceState;

END_STRUCT
END_TYPE

// ---- DUTs/GVL/Inputs/Universal/ST_INPUTS_Unit_UVFilter.TcDUT
TYPE ST_INPUTS_Unit_UVFilter:
STRUCT
	
	Mode:     		E_DeviceMode;
	Command:     E_DeviceState;

END_STRUCT
END_TYPE

// ---- DUTs/GVL/Inputs/Universal/ST_INPUTS_ValveOnOFF.TcDUT
TYPE ST_INPUTS_ValveOnOFF:
STRUCT
	
	Mode:     	E_DeviceMode;
	Command:     E_DeviceState;

END_STRUCT
END_TYPE

// ---- DUTs/GVL/Inputs/Water Treatment/ST_INPUTS_WaterTreatment.TcDUT
TYPE ST_INPUTS_WaterTreatment :
STRUCT

	
	Pump_CleanWaterPumpSelection_A_1_B_0: UINT;
	Pump_WasteWaterSumpPumpSelection_A_1_B_0: UINT;	
	Dosing_Pressure_LOW_Limit: UINT;
	Dosing_Pressure_HIGH_Limit: UINT;

	stWaterQuality: ST_INPUTS_WaterTreatment_Water;
	stSequenceManager: ST_INPUTS_SequenceManager_DM;
	stDosingPump_phUp: ST_INPUTS_DosingPump;
	stDosingPump_phDown: ST_INPUTS_DosingPump;	
	stPump_CleanWaterPumpA: ST_INPUTS_PumpVSD;
	stPump_CleanWaterPumpB: ST_INPUTS_PumpVSD;
	stPump_WasteWaterSumpPumpA : ST_INPUTS_PumpDOL;
	stPump_WasteWaterSumpPumpB : ST_INPUTS_PumpDOL;
	stUnit_OzoneGenerator: ST_INPUTS_Unit_OzoneGenerator;
	stDrumFilter: ST_INPUTS_DrumFilter;
	stUnit_RO_EDI: ST_INPUTS_Unit_RO_EDI;
	stValve_DosingSupply: ST_INPUTS_ValveOnOFF;
	stValve_DM1_Supply: ST_INPUTS_ValveOnOFF;
	stValve_DM2_Supply: ST_INPUTS_ValveOnOFF;
	stValve_Seedling_Stack: ST_INPUTS_ValveOnOFF;
	stValve_SDR_Machine: ST_INPUTS_ValveOnOFF;
	stValve_Tray_Cleaning: ST_INPUTS_ValveOnOFF;
	stValve_FogMisting: ST_INPUTS_ValveOnOFF;
	stValve_TownWater: ST_INPUTS_ValveOnOFF;
	stControlLoopDosing_PH: ST_INPUTS_Dosing_ControlLoop;


	
END_STRUCT
END_TYPE

// ---- DUTs/GVL/Inputs/Water Treatment/ST_INPUTS_WaterTreatment_Water.TcDUT
TYPE ST_INPUTS_WaterTreatment_Water :
STRUCT
	
	PH_LOW_Limit:   UINT;
	PH_HIGH_Limit:  UINT;
	PH_SetPoint:    UINT;
	PH_Selection:   UINT;
	Calibrate_PH: BOOL;
	
	Temp_LOW_Limit:    UINT;
	Temp_HIGH_Limit:    UINT;
	Temp_SetPoint:    UINT;
	Temp_Selection:    UINT;
	Calibrate_Temp: BOOL;


END_STRUCT
END_TYPE

// ---- DUTs/Machines/E_MachineState.TcDUT
{attribute 'qualified_only'}
{attribute 'strict'}
TYPE E_MachineState :
(
	IDLE,
	STARTING,
	RUNNING,
	STOPPING,
	FAULTED
);
END_TYPE

// ---- DUTs/Machines/ST_DMComponents.TcDUT
(*
		This structure is used enable efficient passing device FBs by reference to sub-FBs of the 
		machine FB, while maintaining an instance of each plant component at the 
		highest heirarchy level within the machine FB 
*)

TYPE ST_DMComponents :
STRUCT
	(*
					ACTUATORS (devices that can perform an action)
	*)	

	// Actuated Valves
	fbValve_DosingSupply: 		POINTER TO FB_Valve_ONOFF_woMonitoring;
	fbValve_IrrigatorSupply: 	POINTER TO FB_Valve_ONOFF_woMonitoring; 
	fbValve_WasteWaterReturn: 	POINTER TO FB_Valve_ONOFF_woMonitoring;
	fbValve_DrumFilterRinse: 	POINTER TO FB_Valve_ONOFF_woMonitoring;
	
	// Vendor Units	
	fbUnit_OxyInjector: 		POINTER TO FB_OxygenInjector;	

	// VSD Pumps
	fbPump_MainPumpA: POINTER TO FB_PumpVSD_DanfossFC202;	 
	fbPump_MainPumpB: POINTER TO FB_PumpVSD_DanfossFC202;	 	 
	
	// Filters and Cleaners
	//fbDrumFilter1:				POINTER TO FB_DrumFilter_Faivre120;
	fbUnit_UltraSonCleaner: 	POINTER TO FB_UltraSonicCleaner;
	fbUVFilter1:				POINTER TO FB_UVFilter_UltraAqua_MR4_220PP;
	fbStrainer:					POINTER TO FB_AutoClean_Filter_Bollfilter;
	
	// Passive Components
	fbSumpDosing: 				POINTER TO FB_Tank;
	
	// Dosing Pumps
	fbDosingPump_phUp : POINTER TO FB_DosingPumpPRISMA;
	fbDosingPump_phDown : POINTER TO FB_DosingPumpPRISMA;
	fbDosingPump_NutrientA	: POINTER TO FB_DosingPumpPRISMA;	
	fbDosingPump_NutrientB	: POINTER TO FB_DosingPumpPRISMA;
	fbDosingPump_NutrientC	: POINTER TO FB_DosingPumpPRISMA;
	
	(*
					SENSORS (devices that measure)

	*)	
	// Atlas Sensors
	fbSensor_DissOx1: POINTER TO FB_Sensor_AtlasDO;
	fbSensor_DissOx2: POINTER TO FB_Sensor_AtlasDO;
	fbSensor_DissOx:  POINTER TO FB_DualRedundantSensor;
	
	fbSensor_EC1: POINTER TO FB_Sensor_AtlasEC;
	fbSensor_EC2: POINTER TO FB_Sensor_AtlasEC;
	fbSensor_EC:  POINTER TO FB_DualRedundantSensor;
	
	fbSensor_ORP1: POINTER TO FB_Sensor_AtlasORP;
	fbSensor_ORP2: POINTER TO FB_Sensor_AtlasORP;
	fbSensor_ORP:  POINTER TO FB_DualRedundantSensor;
	
	fbSensor_PH1: POINTER TO FB_Sensor_AtlasPH;
	fbSensor_PH2: POINTER TO FB_Sensor_AtlasPH;
	fbSensor_PH:  POINTER TO FB_DualRedundantSensor;
	
	fbSensor_TMP1: POINTER TO FB_Sensor_AtlasTEMP;
	fbSensor_TMP2: POINTER TO FB_Sensor_AtlasTEMP;
	fbSensor_TMP:  POINTER TO FB_DualRedundantSensor;
	
	fbSensor_SumpLIT1: POINTER TO FB_Sensor_4_20mA_Generic;
	fbSensor_SumpLIT2: POINTER TO FB_Sensor_4_20mA_Generic;
	fbSensor_SumpLIT:  POINTER TO FB_DualRedundantSensor;
 
	fbSensor_FilterPIT1: POINTER TO FB_Sensor_IFM_PG2453;
	fbSensor_FilterPIT2: POINTER TO FB_Sensor_IFM_PG2453;
	fbSensor_DosingPIT1: POINTER TO FB_Sensor_IFM_PG2453;
	
	// Nutrient Tanks
	fbTank_pHUP: POINTER TO FB_Tank;
	fbTank_pHDown: POINTER TO FB_Tank;
	fbTank_NutrientA: POINTER TO FB_Tank;
	fbTank_NutrientB: POINTER TO FB_Tank;
	fbTank_NutrientC: POINTER TO FB_Tank;

	(*
				CONTROL LOOPS (an algorithm that uses sensor data to compute which commans should be sent to actuators)

	*)
		
	// Control Loops
	fbControlLoop_Dosing: POINTER TO FB_ControlLoop_Dosing;
	// fbControlLoop_LevelControl:       <---- in development
	

END_STRUCT
END_TYPE

// ---- DUTs/Machines/ST_POPComponents.TcDUT
(*
		This structure is used enable efficient passing device FBs by reference to sub-FBs of the 
		machine FB, while maintaining an instance of each plant component at the 
		highest heirarchy level within the machine FB 
*)

TYPE ST_POPComponents :
STRUCT
	(*
					ACTUATORS (devices that can perform an action)
	*)	
	// Linear Actuators for vertical movement (POPPING)
	fbLinAct_POP1: 		POINTER TO FB_LinearActuator_Elec;
	fbLinAct_POP2: 		POINTER TO FB_LinearActuator_Elec;
	fbLinAct_POP3: 		POINTER TO FB_LinearActuator_Elec; 
	
	fbStaticConv_POP1: POINTER TO FB_StaticConveyor;
	fbStaticConv_POP2: POINTER TO FB_StaticConveyor;
	fbStaticConv_POP3: POINTER TO FB_StaticConveyor;
	
	fbTrayCentre_POP1: POINTER TO FB_LinearActuator_Pneumatic;
	fbTrayCentre_POP2: POINTER TO FB_LinearActuator_Pneumatic;
	fbTrayCentre_POP3: POINTER TO FB_LinearActuator_Pneumatic;
	
	fbTrayEndSensor: POINTER TO FB_Sensor_OMRON_E3AS;
	
	fbHandshakeUpstream: 	POINTER TO FB_HandShake_TrayMovement;
	fbHandshakeDownstream: 	POINTER TO FB_HandShake_TrayMovement;
	
	
END_STRUCT
END_TYPE

// ---- DUTs/Machines/ST_LFTComponents.TcDUT
(*
		This structure is used enable efficient passing device FBs by reference to sub-FBs of the 
		machine FB, while maintaining an instance of each plant component at the 
		highest heirarchy level within the machine FB 
*)

TYPE ST_LFTComponents :
STRUCT

	fbServo_Lift: 				POINTER TO FB_Lift;
	fbServo_LiftArm: 			POINTER TO FB_LiftArm;
	fbSensor_PressSwitch: 		POINTER TO FB_AutoSwitch();
	fbSensor_Lift_Home: 		POINTER TO FB_AutoSwitch();
	fbSensor_Lift_Top: 			POINTER TO 	FB_AutoSwitch();
	fbSensor_Lift_Bottom: 		POINTER TO FB_AutoSwitch();
	fbSensor_LiftArm_Home: 		POINTER TO 	FB_AutoSwitch();
	fbSensor_LiftArm_Extended: 	POINTER TO 	FB_AutoSwitch();
	fbSensor_LiftArmVacuum:		POINTER TO FB_AutoSwitch();
	fbSensor_LiftBrake_Left: 	POINTER TO FB_AutoSwitch();
	fbSensor_LiftBrake_Right:	POINTER TO FB_AutoSwitch();
	fbAutoGreaser: 				POINTER TO FB_AutoGreaser();
	fbValve_Brake:	 			POINTER TO 	FB_Valve_ONOFF_woMonitoring;
	fbValve_Vacuum: 			POINTER TO 	FB_Valve_ONOFF_woMonitoring;
		
	
	
END_STRUCT
END_TYPE

// ---- DUTs/Machines/ST_RNDDMComponents.TcDUT
(*
		This structure is used enable efficient passing device FBs by reference to sub-FBs of the 
		machine FB, while maintaining an instance of each plant component at the 
		highest heirarchy level within the machine FB 
*)

TYPE ST_RNDDMComponents :
STRUCT
	(*
					ACTUATORS (devices that can perform an action)
	*)	
	// Actuated Valves
	fbValve_RevOsSupply: 		POINTER TO FB_Valve_ONOFF_woMonitoring;
	fbValve_IrrigatorSupply: 	POINTER TO FB_Valve_ONOFF_woMonitoring;
	fbValve_Drain: 	POINTER TO FB_Valve_ONOFF_woMonitoring; 
	// DOL Pump
	fbPump_MainPumpA: 			POINTER TO FB_PumpDOL_Onga413;
	
	// Filters and Cleaners
	fbUVFilter1:				POINTER TO FB_UVFilter_Pentair_EU40;
	
	// Passive Components
	fbSumpDosing: 				POINTER TO FB_Tank;
	
	// Tanks
	fbDosingPump_phUp : 		POINTER TO FB_DosingPumpAgrowtek;
	fbDosingPump_phDown : 		POINTER TO FB_DosingPumpAgrowtek;
	fbDosingPump_NutrientA	: 	POINTER TO FB_DosingPumpAgrowtek;	
	fbDosingPump_NutrientB	: 	POINTER TO FB_DosingPumpAgrowtek;
	fbDosingPump_NutrientC	: 	POINTER TO FB_DosingPumpAgrowtek;
	
	(*
					SENSORS (devices that measure)
	*)	
	fbSensor_DissOx1: 	POINTER TO FB_Sensor_AtlasDO;
	fbSensor_EC1: 		POINTER TO FB_Sensor_AtlasEC;
	fbSensor_ORP1: 		POINTER TO FB_Sensor_AtlasORP;
	fbSensor_PH1: 		POINTER TO FB_Sensor_AtlasPH;
	fbSensor_TMP1: 		POINTER TO FB_Sensor_AtlasTEMP;
	fbSensor_SumpLSH:				POINTER TO FB_Sensor_SICKLevelSwitch_GRF18S;
	
	fbSensor_TankpHUP_LS1:			POINTER TO FB_Sensor_SICKLevelSwitch_GRF18S;
	fbSensor_TankpHDown_LS1:		POINTER TO FB_Sensor_SICKLevelSwitch_GRF18S;
	fbSensor_TankNutrientA_LS1:		POINTER TO FB_Sensor_SICKLevelSwitch_GRF18S;
	fbSensor_TankNutrientB_LS1:		POINTER TO FB_Sensor_SICKLevelSwitch_GRF18S;
	fbSensor_TankNutrientC_LS1:		POINTER TO FB_Sensor_SICKLevelSwitch_GRF18S;
 
	fbSensor_FilterPIT1: POINTER TO FB_Sensor_IFM_PG2453;
	fbSensor_FilterPIT2: POINTER TO FB_Sensor_IFM_PG2453;
	fbSensor_DosingPIT1: POINTER TO FB_Sensor_IFM_PG2453;
	
	// Nutrient Tanks
	fbTank_pHUP: POINTER TO FB_Tank;
	fbTank_pHDown: POINTER TO FB_Tank;
	fbTank_NutrientA: POINTER TO FB_Tank;
	fbTank_NutrientB: POINTER TO FB_Tank;
	fbTank_NutrientC: POINTER TO FB_Tank;
	
	fbUnit_OxyInjector: POINTER TO FB_OxygenInjector;
	(*
				CONTROL LOOPS (an algorithm that uses sensor data to compute which commans should be sent to actuators)
	*)
	// Control Loops
	fbControlLoop_Dosing: POINTER TO FB_ControlLoop_Dosing;
	
	
	fbControlLoop_TankLevel: 	POINTER TO FB_ControlLoop_TankLevel;
	fbControlLoop_DissOx: 		POINTER TO FB_ControlLoop_DissOx;
	
	
	
END_STRUCT
END_TYPE

// ---- DUTs/Machines/ST_RNDWTRComponents.TcDUT
TYPE ST_RNDWTRComponents :
STRUCT
	
	
	// Pumps
	fbPump_CleanWaterPumpA: POINTER TO  FB_PumpDOL_Onga413_RND;

	// Actuator Units
	fbUnit_RO_EDI: POINTER TO FB_Unit_RO_RND;
	
	
	
	// Sensors - Clean Water Tank A (CWT-A) 
	fbSensor_CWT_A_LIT : POINTER TO  FB_Sensor_4_20mA_Generic;
	fbSensor_CWT_A_LSLL : POINTER TO  FB_Sensor_SICKLevelSwitch_GRF18S;
	fbSensor_CWT_A_LSL : POINTER TO  FB_Sensor_SICKLevelSwitch_GRF18S;
	fbSensor_CWT_A_LSH : POINTER TO  FB_Sensor_SICKLevelSwitch_GRF18S;
	fbSensor_CWT_A_LSHH : POINTER TO  FB_Sensor_SICKLevelSwitch_GRF18S;
	
	// Actuated Valves - Incoming
	fbValve_TownWaterSupply: POINTER TO  FB_Valve_ONOFF_woMonitoring;
	
	// Actuated Valves - Outgoing
	fbValve_DM1Supply: POINTER TO  FB_Valve_ONOFF_woMonitoring;
	
	
	// Tanks and Sumps
	fbTank_CWTA: POINTER TO   FB_Tank;
	

END_STRUCT
END_TYPE

// ---- DUTs/Machines/ST_WTRComponents.TcDUT
TYPE ST_WTRComponents :
STRUCT
	// Dosing Pumps
	fbDosingPump_phUp: POINTER TO FB_DosingPumpPRISMA;
	fbDosingPump_phDown: POINTER TO FB_DosingPumpPRISMA;
	
	// Pumps - VSD
	fbPump_CleanWaterPumpA: POINTER TO  FB_PumpVSD_GrundfosCUE;
	fbPump_CleanWaterPumpB: POINTER TO  FB_PumpVSD_GrundfosCUE;
	
	// Pumps - DOL
	fbPump_WasteWaterSumpPumpA : POINTER TO  FB_PumpDOL_Onga413_RND;
	fbPump_WasteWaterSumpPumpB : POINTER TO  FB_PumpDOL_Onga413_RND;
	
	// Actuator Units
	fbUnit_OzoneGenerator: POINTER TO  FB_OzoneGenerator;
	fbDrumFilter_WasteWaterSump: POINTER TO  FB_DrumFilter_Faivre60;
	fbUnit_RO_EDI: POINTER TO FB_Unit_RO_RND;
	
	
	// Sensors - Water PH and Temp
	fbSensor_PH1: POINTER TO  FB_Sensor_AtlasPH;
	fbSensor_PH2: POINTER TO  FB_Sensor_AtlasPH;
	fbSensor_PH: POINTER TO  FB_DualRedundantSensor;
	
	fbSensor_TMP1: POINTER TO  FB_Sensor_AtlasTEMP;
	fbSensor_TMP2: POINTER TO  FB_Sensor_AtlasTEMP;
	fbSensor_TMP: POINTER TO  FB_DualRedundantSensor;
	
	// Sensors - Clean Water Tank A (CWT-A) 
	fbSensor_CWT_A_LIT1 : POINTER TO  FB_Sensor_4_20mA_Generic; 
	fbSensor_CWT_A_LIT2 : POINTER TO  FB_Sensor_4_20mA_Generic;
	fbSensor_CWT_A_LIT : POINTER TO  FB_DualRedundantSensor;
	
	fbSensor_CWT_A_LSLL : POINTER TO  FB_Sensor_SICKLevelSwitch_GRF18S;
	fbSensor_CWT_A_LSL : POINTER TO  FB_Sensor_SICKLevelSwitch_GRF18S;
	fbSensor_CWT_A_LSH : POINTER TO  FB_Sensor_SICKLevelSwitch_GRF18S;
	fbSensor_CWT_A_LSHH : POINTER TO  FB_Sensor_SICKLevelSwitch_GRF18S;
	
	// Sensors - Clean Water Tank B (CWT-B)
	fbSensor_CWT_B_LIT1 : POINTER TO  FB_Sensor_4_20mA_Generic; 
	fbSensor_CWT_B_LIT2 : POINTER TO  FB_Sensor_4_20mA_Generic;
	fbSensor_CWT_B_LIT : POINTER TO  FB_DualRedundantSensor;
	
	fbSensor_CWT_B_LSLL : POINTER TO  FB_Sensor_SICKLevelSwitch_GRF18S;
	fbSensor_CWT_B_LSL : POINTER TO  FB_Sensor_SICKLevelSwitch_GRF18S;
	fbSensor_CWT_B_LSH : POINTER TO  FB_Sensor_SICKLevelSwitch_GRF18S;
	fbSensor_CWT_B_LSHH : POINTER TO  FB_Sensor_SICKLevelSwitch_GRF18S;
	
	// Sensors - Waster Water Sump
	fbSensor_WWS_LSLL : POINTER TO  FB_Sensor_SICKLevelSwitch_GRF18S;
	fbSensor_WWS_LSL : POINTER TO  FB_Sensor_SICKLevelSwitch_GRF18S;
	fbSensor_WWS_LSH : POINTER TO  FB_Sensor_SICKLevelSwitch_GRF18S;
	
	// Sensors - Waster Water Tank
	fbSensor_WWT_LIT1 : POINTER TO  FB_Sensor_4_20mA_Generic; 
	fbSensor_WWT_LIT2 : POINTER TO  FB_Sensor_4_20mA_Generic;
	fbSensor_WWT_LIT : POINTER TO  FB_DualRedundantSensor;
	
	// Actuated Valves - Incoming
	fbValve_TownWaterSupply: POINTER TO  FB_Valve_ONOFF_woMonitoring;
	
	// Actuated Valves - Recirc
	fbValve_DosingSupply: POINTER TO  FB_Valve_ONOFF_woMonitoring;
	
	// Actuated Valves - Outgoing
	fbValve_DM1Supply: POINTER TO  FB_Valve_ONOFF_woMonitoring;
	fbValve_DM2Supply: POINTER TO  FB_Valve_ONOFF_woMonitoring;
	fbValve_SeedStackSupply: POINTER TO  FB_Valve_ONOFF_woMonitoring;
	fbValve_SDRSoakSupply: POINTER TO  FB_Valve_ONOFF_woMonitoring;
	fbValve_WashSupply: POINTER TO  FB_Valve_ONOFF_woMonitoring;
	fbValve_FogMistSupply: POINTER TO  FB_Valve_ONOFF_woMonitoring;
	
	// Tanks and Sumps
	fbTank_CWTA: POINTER TO   FB_Tank;
	fbTank_CWTB: POINTER TO   FB_Tank;
	fbTank_WWT: POINTER TO   FB_Tank;
	fbSump_WWS: POINTER TO   FB_Tank;

END_STRUCT
END_TYPE

// ---- DUTs/ST_INPUTS_LinAct.TcDUT
TYPE ST_INPUTS_LinAct:
STRUCT
	
	Mode:     	E_DeviceMode;
	Command:    E_DeviceState;

END_STRUCT
END_TYPE

// ---- DUTs/ST_INPUTS_POP.TcDUT
TYPE ST_INPUTS_POP:
STRUCT


	stLinAct_POP1: 					ST_INPUTS_LinAct;
	stLinAct_POP2: 					ST_INPUTS_LinAct;
	stLinAct_POP3: 					ST_INPUTS_LinAct;
	
	stStaticConv_POP1:				ST_INPUTS_StaticConv;
	stStaticConv_POP2:				ST_INPUTS_StaticConv;
	stStaticConv_POP3:				ST_INPUTS_StaticConv;
	
	stTrayCentre_POP1:				ST_INPUTS_TrayCentre;
	stTrayCentre_POP2:				ST_INPUTS_TrayCentre;
	stTrayCentre_POP3:				ST_INPUTS_TrayCentre;
	
	stSequenceManager:				ST_INPUTS_SequenceManager_POP;
	
	
	stHandshakeUpstream:			ST_TrayExchangeHandshake;
	stHandshakeDownstream:			ST_TrayExchangeHandshake;
	
	bParamsInitialised: BOOL := FALSE;
	

END_STRUCT
END_TYPE

// ---- DUTs/ST_INPUTS_LFT.TcDUT
TYPE ST_INPUTS_LFT:
STRUCT


	stLinAct_POP1: 					ST_INPUTS_LinAct;
	stLinAct_POP2: 					ST_INPUTS_LinAct;
	stLinAct_POP3: 					ST_INPUTS_LinAct;
	
	stStaticConv_POP1:				ST_INPUTS_StaticConv;
	stStaticConv_POP2:				ST_INPUTS_StaticConv;
	stStaticConv_POP3:				ST_INPUTS_StaticConv;
	
	stTrayCentre_POP1:				ST_INPUTS_TrayCentre;
	stTrayCentre_POP2:				ST_INPUTS_TrayCentre;
	stTrayCentre_POP3:				ST_INPUTS_TrayCentre;
	
	stSequenceManager:				ST_INPUTS_SequenceManager_POP;
	
	
	stHandshakeUpstream:			ST_TrayExchangeHandshake;
	stHandshakeDownstream:			ST_TrayExchangeHandshake;
	
	bParamsInitialised: BOOL := FALSE;
	

END_STRUCT
END_TYPE

// ---- DUTs/ST_INPUTS_SequenceManager_POP.TcDUT
TYPE ST_INPUTS_SequenceManager_POP:
STRUCT
	
	Sequence_Previous: E_SequenceList_RND_DM; // used for resuming previous sequence after calibrartion
	Sequence_Selected: E_SequenceList_RND_DM;
	Sequence_Command: E_SequenceState;
	Sequence_Ack_Interlock: BOOL;
	
	
END_STRUCT
END_TYPE

// ---- DUTs/ST_INPUTS_StaticConv.TcDUT
TYPE ST_INPUTS_StaticConv:
STRUCT
	
	Mode:     	E_DeviceMode;
	Command:    E_DeviceState;

END_STRUCT
END_TYPE

// ---- DUTs/ST_INPUTS_TrayCentre.TcDUT
TYPE ST_INPUTS_TrayCentre:
STRUCT
	
	Mode:     	E_DeviceMode;
	Command:    E_DeviceState;

END_STRUCT
END_TYPE

// ---- DUTs/Universal/E_AlarmPriority.TcDUT
{attribute 'qualified_only'}
{attribute 'strict'}
TYPE E_AlarmPriority :
(
	Diagnostic := 0,
	Low := 1,
	Medium := 2,
	High := 3,
	Critical := 4
);
END_TYPE

// ---- DUTs/Universal/E_DeviceMode.TcDUT
{attribute 'qualified_only'}
{attribute 'strict'}
TYPE E_DeviceMode :
(
	AUTO,
	MANUAL,
	BYPASS,
	SIMULATION
);
END_TYPE

// ---- DUTs/Universal/E_InterlockType.TcDUT
{attribute 'qualified_only'}
{attribute 'strict'}
TYPE E_InterlockType :
(
	RunInterlock,
	StartPermissive,
	StopPermissive
);
END_TYPE

// ---- DUTs/Universal/E_Job_Status.TcDUT
{attribute 'qualified_only'}
{attribute 'strict'}
TYPE E_Job_Status :
(
	waiting := 1,
	placed :=2,
	in_process := 3,
	finished := 4,
	stopped := 5,
	error := 6,
	cancelled := 7
);
END_TYPE

// ---- DUTs/Universal/E_POP_Type.TcDUT
{attribute 'qualified_only'}
{attribute 'strict'}
TYPE E_POP_Type :
(
	EXTEND_CONVEY := 0,
	CONVEY_EXTEND := 1,
	RETRACT_CONVEY := 2,
	CONVEY_RETRACT := 3
);
END_TYPE

// ---- DUTs/Universal/E_SensorType.TcDUT
{attribute 'qualified_only'}
{attribute 'strict'}
TYPE E_SensorType :
(
	Analogue,
	Digital,
	Level
);
END_TYPE

// ---- DUTs/Universal/E_SequenceList_DM.TcDUT
{attribute 'qualified_only'}
{attribute 'strict'}
TYPE E_SequenceList_DM :
(
	SEQ_MAIN := 1,
	SEQ_CALIBRATE := 2,
	SEQ_FILL := 3,
	SEQ_DRAIN := 4
);
END_TYPE

// ---- DUTs/Universal/E_SequenceList_POP.TcDUT
{attribute 'qualified_only'}
{attribute 'strict'}
TYPE E_SequenceList_POP :
(
	SEQ_EXTEND_CONVEY := 1,
	SEQ_CONVEY_EXTEND := 2,
	SEQ_RETRACT_CONVEY := 3,
	SEQ_CONVEY_RETRACT := 4,
	SEQ_EXTEND := 5,
	SEQ_RETRACT := 6
);
END_TYPE

// ---- DUTs/Universal/E_SequenceList_RND_DM.TcDUT
{attribute 'qualified_only'}
{attribute 'strict'}
TYPE E_SequenceList_RND_DM :
(
	SEQ_MAIN := 1,
	SEQ_CALIBRATE := 2,
	SEQ_FILL := 3,
	SEQ_DRAIN := 4,
	SEQ_FLUSH := 5
);
END_TYPE

// ---- DUTs/Universal/E_SequenceList_WTR.TcDUT
{attribute 'qualified_only'}
{attribute 'strict'}
TYPE E_SequenceList_WTR :
(
	SEQ_MAIN := 0,
	SEQ_CALIBRATE := 1
);
END_TYPE

// ---- DUTs/Universal/E_SequenceState.TcDUT
{attribute 'qualified_only'}
{attribute 'strict'}
TYPE E_SequenceState :
(
	RUN,
	STARTING,
	STOP,
	STOPPING,
	HOLD,
	WAIT,
	COMPLETE
);
END_TYPE

// ---- DUTs/Universal/ST_Alarm.TcDUT
TYPE ST_Alarm :
STRUCT
	ePriority: E_AlarmPriority; 
	sLabel: STRING(255);
	bEnabled: BOOL := FALSE;
END_STRUCT
END_TYPE

// ---- DUTs/Universal/ST_Crop.TcDUT
TYPE ST_Crop :
STRUCT
	crop_id : INT;
	crop_status : INT;
	level : INT;
	plant_id : INT;
	stack : INT;
	stage : INT;
	plant : ST_PlantConfig;
END_STRUCT
END_TYPE

// ---- DUTs/Universal/ST_CropJob.TcDUT
TYPE ST_CropJob :
STRUCT
	crop_id : INT;
	datetime_completed : DATE;
	datetime_required : DATE;
	job_id : INT;
	job_status : INT;
	job_type : INT;
	level : INT;
	stack : INT;
	crop : ST_Crop;
END_STRUCT
END_TYPE

// ---- DUTs/Universal/ST_HandShake_TrayMovement.TcDUT
TYPE ST_HandShake_TrayMovement :
STRUCT

	
	
END_STRUCT
END_TYPE

// ---- DUTs/Universal/ST_HVAC.TcDUT
TYPE ST_HVAC :
STRUCT
	Power: BOOL;
	Setpoint: REAL;
END_STRUCT
END_TYPE

// ---- DUTs/Universal/ST_Interlock.TcDUT
TYPE ST_Interlock :
STRUCT
	Active:			BOOL := FALSE;
	Bridge:			BOOL := FALSE;
	
	SubjectDevice:		POINTER TO FB_BaseDevice;
	SubjectVarID: 		STRING;
	SubjectState:		E_DeviceState;
	
	Signal:			BOOL := FALSE;
	Description: 	STRING;
	
	HoldSeq:		BOOL := FALSE; // set to TRUE if the interlock should put sequence into HOLD for operator acknowledgement
	InterlockType:	E_InterlockType;

END_STRUCT
END_TYPE

// ---- DUTs/Universal/ST_Modbus_ReadRequest.TcDUT
TYPE ST_Modbus_ReadRequest :
STRUCT
	
	ReadRegsVals: 				ARRAY[1..10] OF WORD;
	SlaveAddress : 				UINT;
	QtyWordsToRead : 			UINT;
	AdrFirstSlaveRegisterRead: 	UINT;
	bRequestCompleted : 		BOOL;
	bRequestAccepted: 			BOOL;
	bError:						BOOL;

END_STRUCT
END_TYPE

// ---- DUTs/Universal/ST_Modbus_WriteRequest.TcDUT
TYPE ST_Modbus_WriteRequest :
STRUCT

	WriteRegVals: 					ARRAY[1..10] OF WORD;
	SlaveAddress : 					UINT;
	QtyWordsToWrite : 				UINT;
	AdrFirstSlaveRegisterWrite : 	UINT;
	bRequestCompleted: 				BOOL;
	bRequestAccepted: 				BOOL;

END_STRUCT
END_TYPE

// ---- DUTs/Universal/ST_OEE.TcDUT
TYPE ST_OEE :
STRUCT
	dtLastReset: DATE_AND_TIME;
	nNumCycles: UDINT;
	nHrsAvailable: REAL;
	nHrsUtilised: REAL;
	nHrsFaulted: REAL;
END_STRUCT
END_TYPE

// ---- DUTs/Universal/ST_PlantConfig.TcDUT
TYPE ST_PlantConfig :
STRUCT
	average_yield : REAL;
	dark_time : INT;
	seedling_time : INT;
	grow_time : INT;
	plant_id : INT;
	plant_type : STRING;
	seed_spacing : INT;	
	trayConfig : ARRAY[0..3] OF ARRAY[0..3] OF INT;
END_STRUCT
END_TYPE

// ---- DUTs/Universal/ST_SequenceStep.TcDUT
TYPE ST_SequenceStep :
STRUCT
	
	Device:	POINTER TO FB_BaseDevice;
	DeviceVarID: STRING;
	Command:	E_DeviceState;
	StepMinDuration: TIME;
	DelayUntilNextStep: TIME;
	WaitForAction: BOOL;
	
END_STRUCT
END_TYPE

// ---- DUTs/Universal/ST_Tray.TcDUT
TYPE ST_Tray :
STRUCT
	crop_id : INT;
	crop_status : INT;
	level : INT;
	plant_id : INT;
	stack : INT;
	stage : INT;
	plant : ST_PlantConfig;
END_STRUCT
END_TYPE

// ---- DUTs/Universal/ST_TrayExchangeHandshake.TcDUT
TYPE ST_TrayExchangeHandshake :
STRUCT
	eState: E_TrayExchangeState;
	
	bDoneReceiver: 	BOOL := FALSE;
	bDoneSender: 	BOOL := FALSE;
	stTrayIncoming: ST_Tray;
	stTrayOutgoing: ST_Tray;
END_STRUCT
END_TYPE

// ---- DUTs/Universal/ST_Tray_1.TcDUT

TYPE ST_Tray_1 :
STRUCT
	{attribute 'OPC.UA.DA' := '1'}
	nCropID : UDINT;
	{attribute 'OPC.UA.DA' := '0'}
	nLineID : UDINT;
	{attribute 'OPC.UA.DA' := '0'}
	nOrderID : UDINT;
	{attribute 'OPC.UA.DA' := '0'}
	nPlantID : UDINT; 
	{attribute 'OPC.UA.DA' := '0'}
	nStack : INT;
	{attribute 'OPC.UA.DA' := '0'}
	nRack : INT;
	{attribute 'OPC.UA.DA' := '0'}
	nLevel : INT;
	{attribute 'OPC.UA.DA' := '0'}
	nRestack : INT;
	
	{attribute 'OPC.UA.DA' := '1'}
	nTrayQuantity: INT;
	{attribute 'OPC.UA.DA' := '1'}
	nTrayNumber: INT;
	
END_STRUCT
END_TYPE

// ---- DUTs/Universal/ST_Tray_2.TcDUT

TYPE ST_Tray_2 :
STRUCT
	{attribute 'OPC.UA.DA' := '1'}
	nCropID : UDINT;
	{attribute 'OPC.UA.DA' := '0'}
	nLineID : UDINT;
	{attribute 'OPC.UA.DA' := '0'}
	nOrderID : UDINT;
	{attribute 'OPC.UA.DA' := '0'}
	nPlantID : UDINT; 
	{attribute 'OPC.UA.DA' := '0'}
	nStack : INT;
	{attribute 'OPC.UA.DA' := '0'}
	nRack : INT;
	{attribute 'OPC.UA.DA' := '0'}
	nLevel : INT;
	{attribute 'OPC.UA.DA' := '0'}
	nRestack : INT;
	
	{attribute 'OPC.UA.DA' := '1'}
	nTrayQuantity: INT;
	{attribute 'OPC.UA.DA' := '1'}
	nTrayNumber: INT;
	
END_STRUCT
END_TYPE

// ---- POUs/LFT/E_AxisNumberCoE.TcDUT
{attribute 'qualified_only'}
{attribute 'strict'}
TYPE E_AxisNumberCoE :
(
	SingleAxis_LeftDoubleAxis := 1,
	RightDoubleAxis := 2
)WORD;
END_TYPE

// ---- POUs/LFT/E_CoEService.TcDUT
{attribute 'qualified_only'}
{attribute 'strict'}
TYPE E_CoEService : 
(
	NoService := 0,	
	CoERead := 1,
	CoEWrite := 2
	
)WORD;
END_TYPE

// ---- POUs/LFT/E_ConfigurationStateCoE.TcDUT
{attribute 'qualified_only'}
{attribute 'strict'}
TYPE E_ConfigurationStateCoE :
(
	ConfigurationComplete := 0,
	Missing_amsEtherCATMaster_NetID := 1,
	Missing_nEtherCATSlave_Address := 2,
	WrongByteSize				:= 3
);
END_TYPE

// ---- POUs/LFT/E_MovidriveB_OpMode.TcDUT
{attribute 'qualified_only'}
{attribute 'strict'}
TYPE E_MovidriveB_OpMode :
(
	JOG_MODE,
	REFERENCING_MODE,
	AUTOMATIC_MODE
);
END_TYPE

// ---- POUs/LFT/ST_StackDestination.TcDUT
TYPE ST_StackDestination :
STRUCT
	nStack: INT;
	nLevel: INT;
END_STRUCT
END_TYPE

// ---- GVLs/GVL.TcGVL
{attribute 'qualified_only'}
VAR_GLOBAL
	
	LinActPOP_Stroke: INT 					:= 350;
	LinActPOP_Lead: INT 					:= 5;
	LinActPOP_AccelMax: INT 				:= 150;
	LinActPOP_VelocityMax: INT 				:= 300;
	LinActPOP_VelocityJog: INT 				:= 75;
	LinActPOP_TimeExtend: TIME 				:= T#2S;
	LinActPOP_TimeRetract: TIME 			:= T#2S;

	
	StaticConvPOP_IntervalDistance: INT 	:= 4000; 
	StaticConvPOP_GearRatio: INT 			:= 12; 
	StaticConvPOP_AccelMax: INT 			:= 150; 
	StaticConvPOP_VelocityMax: INT 			:= 300; 
	StaticConvPOP_VelocityJog: INT 			:= 100; 
	StaticConvPOP_IntervalTimeFWD: TIME		:= T#5S; 
	StaticConvPOP_IntervalTimeREV: TIME		:= T#5S;
	
	TrayCentrePOP_Stroke: INT 				:= 70; 
	TrayCentrePOP_TimeExtend: TIME 			:= T#5S; 
	TrayCentrePOP_TimeRetract: TIME			:= T#5S;
	
	bEnableInterlocks: BOOL 				:= TRUE;
	bAutoUpdateDeviceState: BOOL			:= FALSE;
	
END_VAR

// ---- GVLs/Inputs.TcGVL
{attribute 'qualified_only'}
VAR_GLOBAL
	
		
	{attribute 'OPC.UA.DA' := '1'}
  	{attribute 'OPC.UA.DA.StructuredType' := '1'}
	SLFT:	ST_INPUTS_LFT;
	
	
	
END_VAR

// ---- GVLs/IO_MAPPING.TcGVL
{attribute 'qualified_only'}
VAR_GLOBAL
	
	mcAxis: AXIS_REF;
END_VAR

// ---- GVLs/Safety.TcGVL
{attribute 'qualified_only'}
VAR_GLOBAL
	{attribute 'OPC.UA.DA' := '1'}
	bSafetyErrorAcknowledge AT %Q*: BOOL; 	
	{attribute 'OPC.UA.DA' := '1'}
	bSafety_Run_Stop AT %Q*: BOOL;
	{attribute 'OPC.UA.DA' := '1'}
	bSafety_EStopStatus AT %I*: BOOL;
	{attribute 'OPC.UA.DA' := '1'}
	bSafety_Reset AT %Q*: BOOL;
	
END_VAR

// ---- POUs/00 Interfaces/I_Device.TcIO
INTERFACE I_Device

METHOD disable : BOOL

VAR_INPUT
END_VAR
END_METHOD

METHOD enable : BOOL

VAR_INPUT
END_VAR
END_METHOD

METHOD setMode : BOOL

VAR_INPUT
	Mode: E_DeviceMode;
END_VAR
END_METHOD

END_INTERFACE

// ---- POUs/00 Interfaces/I_Machine.TcIO
INTERFACE I_Machine

METHOD devices_disable_All : BOOL
END_METHOD

METHOD devices_disable_CurrSeq : BOOL
VAR_INPUT
END_VAR
END_METHOD

METHOD devices_enable_All : BOOL
VAR_INPUT
END_VAR
END_METHOD

METHOD devices_enable_CurrSeq : BOOL
VAR_INPUT
END_VAR
END_METHOD

METHOD devices_setAuto_All : BOOL
VAR_INPUT
END_VAR
END_METHOD

METHOD devices_setAuto_CurrSeq : BOOL
VAR_INPUT
END_VAR
END_METHOD

METHOD devices_setManual_All : BOOL
VAR_INPUT
END_VAR
END_METHOD

METHOD devices_setManual_CurrSeq : BOOL
VAR_INPUT
END_VAR
END_METHOD

END_INTERFACE

// ---- POUs/00 Interfaces/I_PumpDosing.TcIO
INTERFACE I_PumpDosing
(*
	This interface standardises the interface to the 2 x types of dosing pumps being used at ARU installation
	If and when other dosing pumps are used in SF installations they shall implement this interface for the program to function correctly 
	Note: the Agrowtek pumps are supplied in a combined unit (i.e. 5 pumps in 1). 
			IN this case, we shall create 5 instances of the relevant dosing pump FB, not 1 instance for the 5 combined pumps.
*)

METHOD disable : BOOL
VAR_INPUT
END_VAR
END_METHOD

METHOD enable : BOOL
VAR_INPUT
END_VAR
END_METHOD

METHOD executeDose : BOOL
VAR_INPUT
	DoseQtyMls: LREAL;
	DoseRateMlph: UINT;
	RequestComplete: 	POINTER TO BOOL;
END_VAR
VAR_OUTPUT
	RequestAccepted: BOOL;
END_VAR
END_METHOD

METHOD setOFF : BOOL
VAR_INPUT
	RequestComplete: 	POINTER TO BOOL;
END_VAR
VAR_OUTPUT
	RequestAccepted: 	BOOL;
END_VAR
END_METHOD

METHOD setON : BOOL
VAR_INPUT
	RateMlph	 : 		UINT;
	RequestComplete: 	POINTER TO BOOL;
END_VAR

VAR_OUTPUT
	RequestAccepted: 	BOOL;
END_VAR
END_METHOD

END_INTERFACE

// ---- POUs/00 Interfaces/I_PumpVSD.TcIO
INTERFACE I_PumpVSD

METHOD FB_init : BOOL
VAR_INPUT
	bInitRetains : BOOL; // if TRUE, the retain variables are initialized (warm start / cold start)
	bInCopyCode : BOOL;  // if TRUE, the instance afterwards gets moved into the copy code (online change)
	
	PumpID: STRING(80);
	PumpDescr: STRING(255);
	
END_VAR
END_METHOD

METHOD getFrequency : REAL
VAR_INPUT
END_VAR
END_METHOD

METHOD setOff : BOOL
VAR_INPUT
END_VAR
END_METHOD

METHOD setOn : BOOL
VAR_INPUT
END_VAR
END_METHOD

METHOD setReference : BOOL
VAR_INPUT
	RefSetPoint: REAL;
END_VAR
END_METHOD

END_INTERFACE

// ---- POUs/00 Interfaces/I_Sensor.TcIO
INTERFACE I_Sensor

METHOD FB_init : BOOL
VAR_INPUT
	bInitRetains : BOOL; // if TRUE, the retain variables are initialized (warm start / cold start)
	bInCopyCode : BOOL;  // if TRUE, the instance afterwards gets moved into the copy code (online change)
	
	SensorID: STRING(80);
	SensorDescr: STRING(255); 
	SensorType: E_SensorType;
END_VAR
END_METHOD

METHOD getType : E_SensorType
VAR_INPUT
END_VAR
END_METHOD

METHOD getValue : REAL
VAR_INPUT
END_VAR
END_METHOD

METHOD write : BOOL
VAR_INPUT
END_VAR
END_METHOD

END_INTERFACE

// ---- POUs/00 Interfaces/I_Sequence.TcIO
INTERFACE I_Sequence

END_INTERFACE

// ---- POUs/00 Interfaces/I_ValveActuated.TcIO
INTERFACE I_ValveActuated

METHOD close : BOOL
VAR_INPUT
END_VAR
END_METHOD

METHOD FB_init : BOOL
VAR_INPUT
	bInitRetains : BOOL; // if TRUE, the retain variables are initialized (warm start / cold start)
	bInCopyCode : BOOL;  // if TRUE, the instance afterwards gets moved into the copy code (online change)
	
	ValveID: STRING(80);
	ValveDescr: STRING(255); 
	
	Normal_State_NC_1_NO_0: BOOL;
	
END_VAR
END_METHOD

METHOD open : BOOL
VAR_INPUT
END_VAR
END_METHOD

END_INTERFACE

// ---- MAIN.TcPOU
PROGRAM MAIN
VAR
	fbLiftServo: 	FB_SEW_MovidriveB;
	fbLiftArmServo:	FB_SEW_MovidriveB;

	{attribute 'OPC.UA.DA' := '1'}
  	{attribute 'OPC.UA.DA.StructuredType' := '1'}
	fbMachine_Lift:	FB_Machine_LFT(ID:= 'SLFT' , Description:= 'Seeder Lift');
	
	
	{attribute 'OPC.UA.DA' := '1'}
  	{attribute 'OPC.UA.DA.StructuredType' := '1'}
	fbHandshake1:			FB_HandShake_TrayMovement();
	
		
	{attribute 'OPC.UA.DA' := '1'}
  	{attribute 'OPC.UA.DA.StructuredType' := '1'}
	fbHandshake2:			FB_HandShake_TrayMovement();
	
	
	tgGreaser: R_TRIG;
	fbTON_Greaser: TON;
	tGreaser: TIME := T#2S;
	bGreaser AT %Q*: BOOL;
	bGreaser2 AT %Q*: BOOL;
END_VAR



fbTON_Greaser(PT := tGreaser);
tgGreaser();

IF tgGreaser.Q THEN
	fbTON_Greaser.IN := TRUE;
	bGreaser := TRUE;
	bGreaser2 := TRUE;
	tgGreaser.CLK := FALSE;
END_IF

IF fbTON_Greaser.Q THEN
	bGreaser := FALSE;
	bGreaser2 := FALSE;
	fbTON_Greaser.IN := FALSE;
END_IF



fbMachine_Lift(stInputs := Inputs.SLFT, fbHandshakeUpstream := fbHandshake1, fbHandshakeDownstream := fbHandshake2);
fbHandshake1(stTrayExchangeInput := Inputs.SLFT.stHandshakeUpstream);
fbHandshake2(stTrayExchangeInput := Inputs.SLFT.stHandshakeDownstream);
fbLiftServo();
fbLiftArmServo();

END_PROGRAM

// ---- POUs/LFT/FB_SEW_MovidriveB.TcPOU
FUNCTION_BLOCK FB_SEW_MovidriveB EXTENDS FB_BaseDevice

VAR_INPUT 
	// PA2 + PA3 TARGET POSITION
	nTargetPosition: DINT;  // User defined units
	// PA4: SETPOINT SPEED
	nSetpointSpeed: INT; // 1/min
	// PA5 + PA6: ACCELERATION RAMP AND DECELERATION RAMP
	tRamp_Accel: TIME; // 16-bit INT - in seconds
	tRamp_Decel: TIME; // 16-bit INT - in seconds
END_VAR


VAR_OUTPUT
	// PE2 + PE3 ACTUAL POSITION
	nActualPosition: DINT;  // User defined units
	//PE4: ACTUAL SPEED
	nActualSpeed: INT; // 1/min
	//PE5: ACTIVE CURRENT
	nActiveCurrent: INT; // % of rated current
	//PE6: UNIT UTILISATION
	nUnitUtilisation: INT; // % I x t
END_VAR

VAR
	// PROCESS OUTPUT DATA 
	// PO1: CONTROL WORD 2
	bSWLimitSwitch: BOOL;
	bModeHigh: BOOL;
	bModeLow: BOOL;
	bJog_Rev: BOOL := FALSE;
	bJog_Fwd: BOOL := FALSE;
	bStart: BOOL;
	bFaultReset: BOOL;
	bParamSet_SwitchOver: BOOL;
	bRampSwitchover: BOOL;
	bHold_Ctrl: BOOL;
	bEnable_Stop: BOOL;
	bEnable_RapidStop: BOOL;
	bController_Inhibit: BOOL;

	//PROCESS INPUT DATA
	
	// PE1 STATUS WORD
	FaultCode: BYTE;
	bLimSwitch_CCW: BOOL;
	bLimSwitch_CW: BOOL;
	bFault: BOOL;
	bBrakeReleased: BOOL;
	bTargetPosReached: BOOL;
	bIPOSReference: BOOL;
	bInverterReady: BOOL;
	bMotorTurning: BOOL;
	
	// PROCESS DATA WORDS to LINK TO DRIVE
	PO1_ProcessOutput_1 AT %Q* : WORD;
	PO2_ProcessOutput_2 AT %Q* : WORD;
	PO3_ProcessOutput_3 AT %Q* : WORD;
	PO4_ProcessOutput_4 AT %Q* : WORD;
	PO5_ProcessOutput_5 AT %Q* : WORD;
	PO6_ProcessOutput_6 AT %Q* : WORD;
	
	PI1_ProcessInput_1 AT %I* : WORD;
	PI2_ProcessInput_2 AT %I* : WORD;
	PI3_ProcessInput_3 AT %I* : WORD;
	PI4_ProcessInput_4 AT %I* : WORD;
	PI5_ProcessInput_5 AT %I* : WORD;
	PI6_ProcessInput_6 AT %I* : WORD;
	
	// Additional Variables
	eOperatingMode: E_MovidriveB_OpMode := E_MovidriveB_OpMode.JOG_MODE;
	
END_VAR

VAR_OUTPUT PERSISTENT 
	bExtending_1_or_Retracting_0: BOOL;
END_VAR

VAR PERSISTENT
	bAbove_1_or_Below_0_HomePos: BOOL;
	eSMState: (INIT, ENABLE, MOVE_TRIG, MOVING, MOVED, STOP, ERROR, RESET) := INIT;
	nGearRation: REAL; 
	nInertia: REAL;
END_VAR

updateInputs();
updateOutputs();


IF nActualPosition > 0 THEN
	bAbove_1_or_Below_0_HomePos := TRUE;
ELSE
	bAbove_1_or_Below_0_HomePos := FALSE;
END_IF

IF eStateTarget = E_DeviceState.EXTENDED THEN
	eSMState := MOVE_TRIG;
END_IF


CASE eSMState OF
	INIT:
		bController_Inhibit := TRUE;
		bHold_Ctrl := TRUE;
		
	ENABLE:
		bController_Inhibit := FALSE;
		bHold_Ctrl := FALSE;
		eState := E_DeviceState.IDLE;
	
	MOVE_TRIG:
		IF bInverterReady AND ( NOT bFault ) THEN
			bModeLow 	:= TRUE;
			bModeHigh 	:= TRUE;
			eSMState := MOVING;
			
			IF nActualPosition < nTargetPosition THEN
				bExtending_1_or_Retracting_0 := TRUE;
			ELSE
				bExtending_1_or_Retracting_0 := FALSE;
			END_IF
			
		ELSE
			eSMState := ERROR;
		END_IF
		
	MOVING:
		eState := E_DeviceState.EXTENDING;
		
		IF bTargetPosReached THEN
			eSMState := MOVED;
		END_IF
		
	MOVED:
		eState := E_DeviceState.EXTENDED;
		eSMState := ENABLE;
		
	STOP:
		bEnable_Stop := TRUE;
			
	
	ERROR:
		IF bFault THEN
			CASE FaultCode OF
				07:
					// Under-voltage
				08:
					// N-monitoring
				10:
					// IPOS-ILLOP
				14:
					// Encoder
				25:
					// EEPROM
				28:
					// Field-bus timeout
				29:
					// Limit switch reached
				31: 
					// TF Sensor
				36:
					// Immediate switch-off
				42: 
					// Lag fault
				94: 
					// EEPROM checksum
			END_CASE
		END_IF
		//
	RESET:
		bFaultReset := TRUE;
		//
END_CASE

METHOD updateInputs : BOOL
VAR_INPUT
END_VAR
FaultCode 			:= INT_TO_BYTE(SHR((PI1_ProcessInput_1 AND 16#F0), 8));
bLimSwitch_CCW 		:= PI1_ProcessInput_1.7;
bLimSwitch_CW 		:= PI1_ProcessInput_1.6;
bFault 				:= PI1_ProcessInput_1.5;
bBrakeReleased		:= PI1_ProcessInput_1.4;
bTargetPosReached 	:= PI1_ProcessInput_1.3;
bIPOSReference 		:= PI1_ProcessInput_1.2;
bInverterReady 		:= PI1_ProcessInput_1.1;
bMotorTurning 		:= PI1_ProcessInput_1.0;
nActualPosition 	:= SHL(PI2_ProcessInput_2, 8) AND PI3_ProcessInput_3;
nActualSpeed 		:= WORD_TO_INT(PI4_ProcessInput_4);
nActiveCurrent 		:= WORD_TO_INT(PI5_ProcessInput_5);
nUnitUtilisation 	:= WORD_TO_INT(PI6_ProcessInput_6);
END_METHOD

METHOD updateOutputs : BOOL
VAR_INPUT
END_VAR
PO1_ProcessOutput_1.15 := bSWLimitSwitch;
PO1_ProcessOutput_1.12 := bModeHigh;
PO1_ProcessOutput_1.11 := bModeLow;
PO1_ProcessOutput_1.10 := bJog_Rev;
PO1_ProcessOutput_1.9 := bJog_Fwd;
PO1_ProcessOutput_1.8 := bStart;
PO1_ProcessOutput_1.6 := bFaultReset;
PO1_ProcessOutput_1.5 := bParamSet_SwitchOver;
PO1_ProcessOutput_1.4 := bRampSwitchover;
PO1_ProcessOutput_1.3 := bHold_Ctrl;
PO1_ProcessOutput_1.2 := bEnable_Stop; 
PO1_ProcessOutput_1.1 := bEnable_RapidStop;
PO1_ProcessOutput_1.0 := bController_Inhibit;

PO2_ProcessOutput_2 := UDINT_TO_WORD(SHR(nTargetPosition AND 16#F0, 8));
PO3_ProcessOutput_3 := UDINT_TO_WORD(nTargetPosition AND 16#0F);

PO4_ProcessOutput_4 := INT_TO_WORD(nSetpointSpeed);

PO5_ProcessOutput_5 := DINT_TO_WORD(TIME_TO_DINT(tRamp_Accel)/1000);
PO6_ProcessOutput_6 := DINT_TO_WORD(TIME_TO_DINT(tRamp_Decel)/1000);
END_METHOD

END_FUNCTION_BLOCK

// ---- POUs/00 Interfaces/FB_BaseDevice.TcPOU
{attribute 'OPC.UA.DA.StructuredType' := '1'}
FUNCTION_BLOCK FB_BaseDevice

VAR
	{attribute 'OPC.UA.DA' := '1'} 
	sID: STRING; // as per P&IDs
	{attribute 'OPC.UA.DA' := '1'} 
	sDescr: STRING;
	{attribute 'OPC.UA.DA' := '1'} 
	sVarID: STRING;
	{attribute 'OPC.UA.DA' := '0'} 
	bBusy: BOOL := FALSE;
	{attribute 'OPC.UA.DA' := '1'} 
	bError: BOOL := FALSE;
	bEnable: BOOL := TRUE;
	{attribute 'OPC.UA.DA' := '1'} 
	eMode: E_DeviceMode := E_DeviceMode.AUTO;
	{attribute 'OPC.UA.DA' := '1'} 
	eState: E_DeviceState := E_DeviceState.IDLE;
	{attribute 'OPC.UA.DA' := '1'} 
	eStateTarget: E_DeviceState := E_DeviceState.IDLE;
	
	{attribute 'OPC.UA.DA' := '0'} 
	fbTONstartTime: TON;
	{attribute 'OPC.UA.DA' := '0'} 
	fbTONstopTime: TON;
	{attribute 'OPC.UA.DA' := '0'} 
	tMaxStartTime: TIME := T#5S;
	{attribute 'OPC.UA.DA' := '0'} 
	tMaxStopTime: TIME := T#5S;
	
	
	
	{attribute 'OPC.UA.DA' := '1'} 
	aErrors: ARRAY[1..10] OF ST_Alarm;	// raiseEvent() method updates Error1 / aErrors[1] only at the moment, must implement a ring buffer with error active checking for full functionality
	

END_VAR

// This is the base class for all devices (actuators and sensors)
// Provides common variables to all instances 
// Note that the I_Device interface provides the common methods for all devices

METHOD disable : BOOL
VAR_INPUT
END_VAR
bEnable := FALSE;
END_METHOD

METHOD enable : BOOL
VAR_INPUT
END_VAR
bEnable := TRUE;
END_METHOD

METHOD getCommand : E_DeviceState
VAR
	
END_VAR
getCommand := eStateTarget;
END_METHOD

METHOD getDescription : STRING
VAR_INPUT
END_VAR
getDescription := sDescr;
END_METHOD

METHOD getID : STRING
VAR_INPUT
END_VAR
getID := sID;
END_METHOD

METHOD getMode : E_DeviceMode
VAR_INPUT
END_VAR
END_METHOD

METHOD getState : E_DeviceState
VAR
	
END_VAR
getState := eState;
END_METHOD

METHOD getVarID : STRING
VAR_INPUT
END_VAR
getVarID := sVarID;
END_METHOD

METHOD inManual : BOOL
VAR_INPUT
END_VAR
IF eMode = E_DeviceMode.MANUAL THEN
	inManual := TRUE;
ELSE
	inManual := FALSE;
END_IF
END_METHOD

METHOD isEnabled : BOOL
VAR_INPUT
END_VAR
IF bEnable = TRUE THEN
	isEnabled := TRUE;
ELSE
	isEnabled := FALSE;
END_IF
END_METHOD

METHOD raiseAlarm : POINTER TO ST_Alarm
VAR_INPUT
	Priority: E_AlarmPriority; 
	Label: STRING(255);
	Enabled: BOOL := FALSE;
	DeviceAlarmID: INT; // from 1 to 10
END_VAR
aErrors[DeviceAlarmID].bEnabled := TRUE;
aErrors[DeviceAlarmID].ePriority := Priority;
aErrors[DeviceAlarmID].sLabel := Label;
END_METHOD

METHOD runSimulation : BOOL
VAR_INPUT
END_VAR
eState := eStateTarget;
END_METHOD

METHOD setCommand : BOOL
VAR_INPUT
	StateTarget: E_DeviceState;
END_VAR
eStateTarget := StateTarget;
END_METHOD

METHOD setID : BOOL
VAR_INPUT
	ID: STRING;
END_VAR
sID := ID;
END_METHOD

METHOD setMode : BOOL
VAR_INPUT
	Mode: E_DeviceMode;
END_VAR

eMode := Mode;
END_METHOD

METHOD setVarID : BOOL
VAR_INPUT
	VarID: STRING;
END_VAR
sVarID := VarID;
END_METHOD

END_FUNCTION_BLOCK

// ---- POUs/06 Machines/FB_Machine_LFT.TcPOU
{attribute 'OPC.UA.DA.StructuredType' := '1'}
FUNCTION_BLOCK FB_Machine_LFT EXTENDS FB_BaseMachine IMPLEMENTS I_Machine



VAR_IN_OUT PERSISTENT
	
	stInputs: ST_INPUTS_LFT;
		
	{attribute 'OPC.UA.DA' := '1'}
  	{attribute 'OPC.UA.DA.StructuredType' := '1'}
	fbHandshakeUpstream: 	FB_HandShake_TrayMovement();
		
	{attribute 'OPC.UA.DA' := '1'}
  	{attribute 'OPC.UA.DA.StructuredType' := '1'}
	fbHandshakeDownstream: 	FB_HandShake_TrayMovement();
	
END_VAR



VAR
	
	stTrayCurrent: ST_Tray;
	
	bIsFirstRun: BOOL := TRUE;
	bEnableIgnitionControl: BOOL := TRUE;
	bFirstInputScan: BOOL := TRUE;
	
	
	{attribute 'OPC.UA.DA' := '1'}
  	{attribute 'OPC.UA.DA.StructuredType' := '1'}
	fbServo_Lift: FB_Lift;
	 					
	

		
	{attribute 'OPC.UA.DA' := '1'}
  	{attribute 'OPC.UA.DA.StructuredType' := '1'}														
	fbServo_LiftArm: FB_LiftArm;
		
	
		
	{attribute 'OPC.UA.DA' := '1'}
  	{attribute 'OPC.UA.DA.StructuredType' := '1'}
	fbSensor_PressSwitch:				FB_AutoSwitch();
		
	{attribute 'OPC.UA.DA' := '1'}
  	{attribute 'OPC.UA.DA.StructuredType' := '1'}
	fbSensor_Lift_Home:					FB_AutoSwitch();
		
	{attribute 'OPC.UA.DA' := '1'}
  	{attribute 'OPC.UA.DA.StructuredType' := '1'}
	fbSensor_Lift_Top:					FB_AutoSwitch();
		
	{attribute 'OPC.UA.DA' := '1'}
  	{attribute 'OPC.UA.DA.StructuredType' := '1'}
	fbSensor_Lift_Bottom:				FB_AutoSwitch();
	
		
	{attribute 'OPC.UA.DA' := '1'}
  	{attribute 'OPC.UA.DA.StructuredType' := '1'}
	fbSensor_LiftArm_Home:				FB_AutoSwitch();
		
	{attribute 'OPC.UA.DA' := '1'}
  	{attribute 'OPC.UA.DA.StructuredType' := '1'}
	fbSensor_LiftArm_Extended:			FB_AutoSwitch();
		
	{attribute 'OPC.UA.DA' := '1'}
  	{attribute 'OPC.UA.DA.StructuredType' := '1'}
	fbSensor_LiftArmVacuum:				FB_AutoSwitch();
		
	{attribute 'OPC.UA.DA' := '1'}
  	{attribute 'OPC.UA.DA.StructuredType' := '1'}
	fbSensor_LiftBrake_Left:			FB_AutoSwitch();
		
	{attribute 'OPC.UA.DA' := '1'}
  	{attribute 'OPC.UA.DA.StructuredType' := '1'}
	fbSensor_LiftBrake_Right:			FB_AutoSwitch();
		
	{attribute 'OPC.UA.DA' := '1'}
  	{attribute 'OPC.UA.DA.StructuredType' := '1'}
	fbAutoGreaser:						FB_AutoGreaser();
		
	{attribute 'OPC.UA.DA' := '1'}
  	{attribute 'OPC.UA.DA.StructuredType' := '1'}
	fbValve_Brake:						FB_Valve_ONOFF_woMonitoring(ValveID:= 'BKV', ValveDescr:= 'Brake Solenoid Valve' , Normal_State_NC_1_NO_0:= TRUE);
		
	{attribute 'OPC.UA.DA' := '1'}
  	{attribute 'OPC.UA.DA.StructuredType' := '1'}
	fbValve_Vacuum:						FB_Valve_ONOFF_woMonitoring(ValveID:= 'VPV', ValveDescr:= 'Vacuum Solenoid Valve' , Normal_State_NC_1_NO_0:= TRUE);
		
	
	
	(**
	**		TESTING / SIMULATION VARIABLES
	**)
	
	tgStartSeq: R_TRIG;
	bExt_Step2: BOOL := FALSE;
	bExt_Step8: BOOL := FALSE;
	bPWR_CTRL AT %Q* : BOOL;
	bLOCK_CTRL AT %Q* : BOOL;
	
END_VAR

VAR PERSISTENT
													
	// Package all components into structure & array 
	// ST used for readability
	// Arrray used for iterability 
	stAllComponents: ST_LFTComponents;
	
		
	{attribute 'OPC.UA.DA' := '1'}
  	{attribute 'OPC.UA.DA.StructuredType' := '1'}
	fbInterlocks: 			FB_InterlockManager;
	
	bInProgress: BOOL := FALSE;	//used as a flag to signify that we are in an operation
	
	// Sequences
	//fbSeq_MOVE: 	FB_SequenceMOVE;

	//aSeqs: ARRAY[1..10] OF FB_SequenceBase;	
	
	// Maglock
	
	
END_VAR

IF bIsFirstRun THEN
	devices_init();
	devices_update();
	//sequence_init();
	bIsFirstRun := FALSE;
END_IF


devices_update();
(*
// Scan inputs from OPC
IF stInputs.bParamsInitialised AND bEnableIgnitionControl THEN
	IF bFirstInputScan THEN
		stInputs.stSequenceManager.Sequence_Selected := 1;
		stInputs.stSequenceManager.Sequence_Command := E_SequenceState.STOP;
		fbSequenceManager.selectSequence(Sequence := 1); // main sequence
		fbSequenceManager.stopSequence();
		bFirstInputScan := FALSE;
	END_IF
	scanOPCInputs(Inputs := stInputs ); // only scan if SCADA has set the imputs, otherwise keep persistent or initalised variables
END_IF

*)
// Sequence manager
// fbSeq_MOVE.populateSteps();
// aSeqs[1] := fbSeq_MOVE;
// fbSequenceManager(aSequences := aSeqs);

// Interlocks (make sure this is always called second last (so it overrides any target states set by the sequence manager)
IF GVL.bEnableInterlocks THEN
	interlocks();
END_IF

// Update devices
devices_update();
handshakes();
// sequence();


(**
**		TESTING / SIMULATION VARIABLES
**)

(*
tgStartSeq();
IF tgStartSeq.Q THEN
	fbSequenceManager.selectSequence(Sequence := 1);
	fbSequenceManager.startSequence();
END_IF
*)

METHOD devices_init : BOOL
VAR
	VarInfo : __SYSTEM.VAR_INFO;
	setVarID: INT;
END_VAR
// Hold References to devices in a structure and also an array
// A structure is useful where devices are accessed by name (handy with auto-complete and readability)
// The array is useful for when we want to iterate through all of the devices in the machine and apply a global command (i.e. disable all devices)

// Extract the function block instance name and insert it to each function block
// This enables us to share only the function block name over OPC for nested instances (i.e. sequences, interlock manager)
// The contents of each function block is shared over OPC within the Machine as per heirarchy
// When Ignition needs to retrieve details of devices at the interlock manager and sequence, it simply performs a lookup using the VarID as a key



VarInfo := __VARINFO(fbServo_Lift);
fbServo_Lift.setVarID(VarID := VarInfo.Symbol);

VarInfo := __VARINFO(fbServo_LiftArm);
fbServo_LiftArm.setVarID(VarID := VarInfo.Symbol);

VarInfo := __VARINFO(fbSensor_PressSwitch);
fbSensor_PressSwitch.setVarID(VarID := VarInfo.Symbol);

VarInfo := __VARINFO(fbSensor_Lift_Home);
fbSensor_Lift_Home.setVarID(VarID := VarInfo.Symbol);

VarInfo := __VARINFO(fbSensor_Lift_Top);
fbSensor_Lift_Top.setVarID(VarID := VarInfo.Symbol);

VarInfo := __VARINFO(fbSensor_Lift_Bottom);
fbSensor_Lift_Bottom.setVarID(VarID := VarInfo.Symbol);

VarInfo := __VARINFO(fbSensor_LiftArm_Home);
fbSensor_LiftArm_Home.setVarID(VarID := VarInfo.Symbol);

VarInfo := __VARINFO(fbSensor_LiftArm_Extended);
fbSensor_LiftArm_Extended.setVarID(VarID := VarInfo.Symbol);

VarInfo := __VARINFO(fbSensor_LiftArmVacuum);
fbSensor_LiftArmVacuum.setVarID(VarID := VarInfo.Symbol);

VarInfo := __VARINFO(fbSensor_LiftBrake_Left);
fbSensor_LiftBrake_Left.setVarID(VarID := VarInfo.Symbol);

VarInfo := __VARINFO(fbSensor_LiftBrake_Right);
fbSensor_LiftBrake_Right.setVarID(VarID := VarInfo.Symbol);

VarInfo := __VARINFO(fbAutoGreaser);
fbAutoGreaser.setVarID(VarID := VarInfo.Symbol);

VarInfo := __VARINFO(fbValve_Brake);
fbValve_Brake.setVarID(VarID := VarInfo.Symbol);

VarInfo := __VARINFO(fbValve_Vacuum);
fbValve_Vacuum.setVarID(VarID := VarInfo.Symbol);

aAllComponents[1]  :=  ADR(fbServo_LifT);
aAllComponents[2]  :=  ADR(fbServo_LiftArm);
aAllComponents[3]  :=  ADR(fbSensor_PressSwitch);
aAllComponents[4]  :=  ADR(fbSensor_Lift_Home );
aAllComponents[5]  :=  ADR(fbSensor_Lift_Top );
aAllComponents[6]  :=  ADR(fbSensor_LiftArm_Home  );
aAllComponents[7]  :=  ADR(fbSensor_LiftArm_Extended );
aAllComponents[8]  :=  ADR(fbSensor_LiftArmVacuum );
aAllComponents[9]  :=  ADR(fbSensor_LiftBrake_Left );
aAllComponents[10]  :=  ADR(fbSensor_LiftBrake_Right);
aAllComponents[11]  :=  ADR(fbAutoGreaser);
aAllComponents[12]  :=  ADR(fbValve_Brake);
aAllComponents[13]  :=  ADR(fbValve_Vacuum);
aAllComponents[14]  :=  ADR(fbHandshakeDownstream);
aAllComponents[15]  :=  ADR(fbHandshakeUpstream);



fbServo_LifT.setID(ID := 'Sample ID');									
fbServo_LiftArm.setID(ID := 'Sample ID');
fbSensor_PressSwitch.setID(ID := 'Sample ID');
fbSensor_Lift_Home.setID(ID := 'Sample ID');			
fbSensor_Lift_Top.setID(ID := 'Sample ID');
fbSensor_Lift_Bottom.setID(ID := 'Sample ID');
fbSensor_LiftArm_Home.setID(ID := 'Sample ID');
fbSensor_LiftArm_Extended.setID(ID := 'Sample ID');
fbSensor_LiftArmVacuum.setID(ID := 'Sample ID');
fbSensor_LiftBrake_Left.setID(ID := 'Sample ID');
fbSensor_LiftBrake_Right.setID(ID := 'Sample ID');
fbAutoGreaser.setID(ID := 'Sample ID');			
fbValve_Brake.setID(ID := 'Sample ID');		
fbValve_Vacuum.setID(ID := 'Sample ID');	
fbHandshakeDownstream.setID(ID := 'Downstream tray exchange handshake');
fbHandshakeUpstream.setID(ID := 'Upstream tray exchange handshake');



stAllComponents.fbServo_Lift 				:= ADR(fbServo_Lift);
stAllComponents.fbServo_LiftArm				:= ADR(fbServo_LiftArm);
stAllComponents.fbSensor_PressSwitch		:= ADR(fbSensor_PressSwitch);
stAllComponents.fbSensor_Lift_Home			:= ADR(fbSensor_Lift_Home);
stAllComponents.fbSensor_Lift_Top			:= ADR(fbSensor_Lift_Top);
stAllComponents.fbSensor_Lift_Bottom		:= ADR(fbSensor_Lift_Bottom);
stAllComponents.fbSensor_LiftArm_Home		:= ADR(fbSensor_LiftArm_Home);
stAllComponents.fbSensor_LiftArm_Extended	:= ADR(fbSensor_LiftArm_Extended);
stAllComponents.fbSensor_LiftArmVacuum		:= ADR(fbSensor_LiftArmVacuum);
stAllComponents.fbSensor_LiftBrake_Left		:= ADR(fbSensor_LiftBrake_Left);
stAllComponents.fbSensor_LiftBrake_Right	:= ADR(fbSensor_LiftBrake_Right);
stAllComponents.fbAutoGreaser				:= ADR(fbAutoGreaser);
stAllComponents.fbValve_Brake				:= ADR(fbValve_Brake);
stAllComponents.fbValve_Vacuum				:= ADR(fbValve_Vacuum);


// Note that the soil sensors have not been added to the stAllComponents or components array at this stage
// They are not being used in sequences or interlocks (at this stage)

nQtyComponents := 15;

devices_disable_All();
END_METHOD

METHOD devices_update : BOOL
VAR_INPUT
END_VAR
fbServo_LifT();									
fbServo_LiftArm();
fbSensor_PressSwitch();
fbSensor_Lift_Home();			
fbSensor_Lift_Top();
fbSensor_Lift_Bottom();
fbSensor_LiftArm_Home();
fbSensor_LiftArm_Extended();
fbSensor_LiftArmVacuum();
fbSensor_LiftBrake_Left();
fbSensor_LiftBrake_Right();
fbAutoGreaser();			
fbValve_Brake();		
fbValve_Vacuum();	
fbHandshakeDownstream();
fbHandshakeUpstream();
END_METHOD

METHOD FB_init : BOOL
VAR_INPUT
	bInitRetains : BOOL; // if TRUE, the retain variables are initialized (warm start / cold start)
	bInCopyCode : BOOL;  // if TRUE, the instance afterwards gets moved into the copy code (online change)
	
	ID: STRING;
	Description: STRING;

	
END_VAR
sID := ID;
sDescr := Description;
END_METHOD

METHOD handshakes : BOOL
VAR_INPUT
END_VAR
(*
*
*				DOWNSTREAM HANDSHAKE (we are sending a tray downstream)
*)

(*

IF fbHandshakeDownstream.stTrayExchgangeOutput.eState = E_TrayExchangeState.IDLE AND (fbSensor_TrayEnd.getState() = E_DeviceState.ON) THEN
	fbHandshakeDownstream.stTrayExchangeInput.eState := E_TrayExchangeState.REQUESTED;
END_IF

IF fbHandshakeDownstream.stTrayExchgangeOutput.eState = E_TrayExchangeState.ACCEPTED THEN //AND bTrayisReady THEN
	fbHandshakeDownstream.stTrayExchangeInput.eState := E_TrayExchangeState.IN_PROGRESS;
END_IF

IF fbHandshakeDownstream.stTrayExchgangeOutput.eState = E_TrayExchangeState.COMPLETED THEN
	fbHandshakeDownstream.stTrayExchangeInput.stTrayOutgoing := stTrayCurrent;
END_IF



(*
*
*				UPSTREAM HANDSHAKE (we are receiving a tray)
*)


IF fbHandshakeUpstream.stTrayExchgangeOutput.eState = E_TrayExchangeState.REQUESTED  THEN // bTrayisReady THEN
	fbHandshakeUpstream.stTrayExchangeInput.eState := E_TrayExchangeState.ACCEPTED;
END_IF


IF fbHandshakeUpstream.stTrayExchgangeOutput.eState = E_TrayExchangeState.ACCEPTED THEN // AND bStartingtoMove THEN
	fbHandshakeUpstream.stTrayExchangeInput.eState := E_TrayExchangeState.IN_PROGRESS;
END_IF


IF fbHandshakeUpstream.stTrayExchgangeOutput.eState = E_TrayExchangeState.COMPLETED THEN
	stTrayCurrent := fbHandshakeUpstream.stTrayExchangeInput.stTrayOutgoing;
END_IF

*)
END_METHOD

METHOD interlocks : BOOL
VAR_INPUT
END_VAR
fbInterlocks.init();

(*
fbInterlocks.update(
							Description:= 'Linear Actuator 1 Attempted to Move While Static Conveyor Running',
							InterlockType:= E_InterlockType.RunInterlock, 
							Subject_Device:= ADR(fbLinAct_POP1), 
							Subject_State:= E_DeviceState.IDLE, 
							Signal:=  (fbStaticConv_POP1.getState() = E_DeviceState.RUNNING) OR (fbStaticConv_POP2.getState() = E_DeviceState.RUNNING)
										OR (fbStaticConv_POP3.getState() = E_DeviceState.RUNNING) OR (fbStaticConv_POP1.getState() = E_DeviceState.REVERSE) OR (fbStaticConv_POP2.getState() = E_DeviceState.REVERSE)
										OR (fbStaticConv_POP3.getState() = E_DeviceState.REVERSE),
							HoldSequence:=	FALSE);
							

fbInterlocks.update(
							Description:= 'Linear Actuator 2 Attempted to Move While Static Conveyor Running',
							InterlockType:= E_InterlockType.RunInterlock, 
							Subject_Device:= ADR(fbLinAct_POP2), 
							Subject_State:= E_DeviceState.IDLE, 
							Signal:=  (fbStaticConv_POP1.getState() = E_DeviceState.RUNNING) OR (fbStaticConv_POP2.getState() = E_DeviceState.RUNNING)
										OR (fbStaticConv_POP3.getState() = E_DeviceState.RUNNING) OR (fbStaticConv_POP1.getState() = E_DeviceState.REVERSE) OR (fbStaticConv_POP2.getState() = E_DeviceState.REVERSE)
										OR (fbStaticConv_POP3.getState() = E_DeviceState.REVERSE),
							HoldSequence:=	FALSE);

fbInterlocks.update(
							Description:= 'Linear Actuator 3 Attempted to Move While Static Conveyor Running',
							InterlockType:= E_InterlockType.RunInterlock, 
							Subject_Device:= ADR(fbLinAct_POP3), 
							Subject_State:= E_DeviceState.IDLE, 
							Signal:=  (fbStaticConv_POP1.getState() = E_DeviceState.RUNNING) OR (fbStaticConv_POP2.getState() = E_DeviceState.RUNNING)
										OR (fbStaticConv_POP3.getState() = E_DeviceState.RUNNING) OR (fbStaticConv_POP1.getState() = E_DeviceState.REVERSE) OR (fbStaticConv_POP2.getState() = E_DeviceState.REVERSE)
										OR (fbStaticConv_POP3.getState() = E_DeviceState.REVERSE),
							HoldSequence:=	FALSE);
							
							
fbInterlocks.update(
							Description:= 'Static Conveyor 1 Attemped to Move While POPs Are Moving',
							InterlockType:= E_InterlockType.RunInterlock, 
							Subject_Device:= ADR(fbStaticConv_POP1), 
							Subject_State:= E_DeviceState.IDLE, 
							Signal:=  (fbLinAct_POP1.getState() = E_DeviceState.RUNNING) OR (fbLinAct_POP2.getState() = E_DeviceState.RUNNING)
										OR (fbLinAct_POP3.getState() = E_DeviceState.RUNNING) OR (fbLinAct_POP1.getState() = E_DeviceState.REVERSE) OR (fbLinAct_POP2.getState() = E_DeviceState.REVERSE)
										OR (fbLinAct_POP3.getState() = E_DeviceState.REVERSE),
							HoldSequence:=	FALSE);
							

fbInterlocks.update(
							Description:= 'Static Conveyor 2 Attemped to Move While POPs Are Moving',
							InterlockType:= E_InterlockType.RunInterlock, 
							Subject_Device:= ADR(fbStaticConv_POP2), 
							Subject_State:= E_DeviceState.IDLE, 
							Signal:=  (fbLinAct_POP1.getState() = E_DeviceState.RUNNING) OR (fbLinAct_POP2.getState() = E_DeviceState.RUNNING)
										OR (fbLinAct_POP3.getState() = E_DeviceState.RUNNING) OR (fbLinAct_POP1.getState() = E_DeviceState.REVERSE) OR (fbLinAct_POP2.getState() = E_DeviceState.REVERSE)
										OR (fbLinAct_POP3.getState() = E_DeviceState.REVERSE),
							HoldSequence:=	FALSE);
							

fbInterlocks.update(
							Description:= 'Static Conveyor 3 Attemped to Move While POPs Are Moving',
							InterlockType:= E_InterlockType.RunInterlock, 
							Subject_Device:= ADR(fbStaticConv_POP3), 
							Subject_State:= E_DeviceState.IDLE, 
							Signal:=  (fbLinAct_POP1.getState() = E_DeviceState.RUNNING) OR (fbLinAct_POP2.getState() = E_DeviceState.RUNNING)
										OR (fbLinAct_POP3.getState() = E_DeviceState.RUNNING) OR (fbLinAct_POP1.getState() = E_DeviceState.REVERSE) OR (fbLinAct_POP2.getState() = E_DeviceState.REVERSE)
										OR (fbLinAct_POP3.getState() = E_DeviceState.REVERSE),
							HoldSequence:=	FALSE);	

							
fbInterlocks.update(
							Description:= 'Static Conveyor 1 Attemped to Move When Tray Centre Actuators are Centred',
							InterlockType:= E_InterlockType.RunInterlock, 
							Subject_Device:= ADR(fbStaticConv_POP1), 
							Subject_State:= E_DeviceState.IDLE, 
							Signal:=  (fbTrayCentre_POP1.getState() = E_DeviceState.EXTENDED) OR (fbTrayCentre_POP2.getState() = E_DeviceState.EXTENDED)
										OR (fbTrayCentre_POP3.getState() = E_DeviceState.EXTENDED),
							HoldSequence:=	FALSE);							
							
fbInterlocks.update(
							Description:= 'Static Conveyor 2 Attemped to Move When Tray Centre Actuators are Centred',
							InterlockType:= E_InterlockType.RunInterlock, 
							Subject_Device:= ADR(fbStaticConv_POP2), 
							Subject_State:= E_DeviceState.IDLE, 
							Signal:=  (fbTrayCentre_POP1.getState() = E_DeviceState.EXTENDED) OR (fbTrayCentre_POP2.getState() = E_DeviceState.EXTENDED)
										OR (fbTrayCentre_POP3.getState() = E_DeviceState.EXTENDED),
							HoldSequence:=	FALSE);		
							
							
fbInterlocks.update(
							Description:= 'Static Conveyor 3 Attemped to Move When Tray Centre Actuators are Centred',
							InterlockType:= E_InterlockType.RunInterlock, 
							Subject_Device:= ADR(fbStaticConv_POP3), 
							Subject_State:= E_DeviceState.IDLE, 
							Signal:=  (fbTrayCentre_POP1.getState() = E_DeviceState.EXTENDED) OR (fbTrayCentre_POP2.getState() = E_DeviceState.EXTENDED)
										OR (fbTrayCentre_POP3.getState() = E_DeviceState.EXTENDED),
							HoldSequence:=	FALSE);		
							
							
							
(* HANDSHAKING INTERLOCKS *)
							
fbInterlocks.update(
							Description:= 'Wait for tray RESQUESTED signal',
							InterlockType:= E_InterlockType.RunInterlock, 
							Subject_Device:= ADR(fbStaticConv_POP1), 
							Subject_State:= E_DeviceState.IDLE, 
							Signal:=  ((fbSequenceManager.getCurrentSeq_ID() = E_SequenceList_POP.SEQ_EXTEND_CONVEY) OR
										(fbSequenceManager.getCurrentSeq_ID() = E_SequenceList_POP.SEQ_RETRACT_CONVEY)) AND
										fbHandshakeDownstream.stTrayExchgangeOutput.eState <> E_TrayExchangeState.IN_PROGRESS,
							HoldSequence:=	FALSE);		
							
							
fbInterlocks.update(
							Description:= 'Wait for tray RESQUESTED signal',
							InterlockType:= E_InterlockType.RunInterlock, 
							Subject_Device:= ADR(fbStaticConv_POP2), 
							Subject_State:= E_DeviceState.IDLE, 
							Signal:=  ((fbSequenceManager.getCurrentSeq_ID() = E_SequenceList_POP.SEQ_EXTEND_CONVEY) OR
										(fbSequenceManager.getCurrentSeq_ID() = E_SequenceList_POP.SEQ_RETRACT_CONVEY)) AND
										fbHandshakeDownstream.stTrayExchgangeOutput.eState <> E_TrayExchangeState.IN_PROGRESS,
							HoldSequence:=	FALSE);		

fbInterlocks.update(
							Description:= 'Wait for tray RESQUESTED signal',
							InterlockType:= E_InterlockType.RunInterlock, 
							Subject_Device:= ADR(fbStaticConv_POP3), 
							Subject_State:= E_DeviceState.IDLE, 
							Signal:=  ((fbSequenceManager.getCurrentSeq_ID() = E_SequenceList_POP.SEQ_EXTEND_CONVEY) OR
										(fbSequenceManager.getCurrentSeq_ID() = E_SequenceList_POP.SEQ_RETRACT_CONVEY)) AND
										fbHandshakeDownstream.stTrayExchgangeOutput.eState <> E_TrayExchangeState.IN_PROGRESS,
							HoldSequence:=	FALSE);									
							
fbInterlocks.update(
							Description:= 'Wait for tray RESQUESTED signal',
							InterlockType:= E_InterlockType.RunInterlock, 
							Subject_Device:= ADR(fbLinAct_POP1), 
							Subject_State:= E_DeviceState.IDLE, 
							Signal:=  ((fbSequenceManager.getCurrentSeq_ID() = E_SequenceList_POP.SEQ_CONVEY_EXTEND) OR
										(fbSequenceManager.getCurrentSeq_ID() = E_SequenceList_POP.SEQ_CONVEY_RETRACT)) AND
										fbHandshakeDownstream.stTrayExchgangeOutput.eState <> E_TrayExchangeState.IN_PROGRESS,
							HoldSequence:=	FALSE);		

fbInterlocks.update(
							Description:= 'Wait for tray RESQUESTED signal',
							InterlockType:= E_InterlockType.RunInterlock, 
							Subject_Device:= ADR(fbLinAct_POP2), 
							Subject_State:= E_DeviceState.IDLE, 
							Signal:=  ((fbSequenceManager.getCurrentSeq_ID() = E_SequenceList_POP.SEQ_CONVEY_EXTEND) OR
										(fbSequenceManager.getCurrentSeq_ID() = E_SequenceList_POP.SEQ_CONVEY_RETRACT)) AND
										fbHandshakeDownstream.stTrayExchgangeOutput.eState <> E_TrayExchangeState.IN_PROGRESS,
							HoldSequence:=	FALSE);									

fbInterlocks.update(
							Description:= 'Wait for tray RESQUESTED signal',
							InterlockType:= E_InterlockType.RunInterlock, 
							Subject_Device:= ADR(fbLinAct_POP3), 
							Subject_State:= E_DeviceState.IDLE, 
							Signal:=  ((fbSequenceManager.getCurrentSeq_ID() = E_SequenceList_POP.SEQ_CONVEY_EXTEND) OR
										(fbSequenceManager.getCurrentSeq_ID() = E_SequenceList_POP.SEQ_CONVEY_RETRACT)) AND
										fbHandshakeDownstream.stTrayExchgangeOutput.eState <> E_TrayExchangeState.IN_PROGRESS,
							HoldSequence:=	FALSE);		

*)
fbInterlocks.execute();
END_METHOD

METHOD scanOPCInputs : BOOL
VAR_INPUT
	Inputs: ST_INPUTS_LFT;
END_VAR

VAR 
	nCurrenSeq_Temp: INT;
	nPrev_Seq: INT;
END_VAR

(*
			SEQUENCE CONTROL
*)



IF stInputs.stSequenceManager.Sequence_Selected <> fbSequenceManager.getCurrentSeq_ID() THEN // Selected sequence has been changed
	fbSequenceManager.stopSequence();
	devices_disable_All();
	fbSequenceManager.selectSequence(stInputs.stSequenceManager.Sequence_Selected);
	devices_enable_CurrSeq();
END_IF


IF stInputs.stSequenceManager.Sequence_Ack_Interlock THEN
	fbSequenceManager.acknowledgePause();
	stInputs.stSequenceManager.Sequence_Ack_Interlock := FALSE;
END_IF


CASE stInputs.stSequenceManager.Sequence_Command OF
	E_SequenceState.RUN:
		IF fbSequenceManager.getState() <> E_SequenceState.RUN THEN
			fbSequenceManager.startSequence();
			stInputs.stSequenceManager.Sequence_Command := E_SequenceState.WAIT;
		END_IF
	E_SequenceState.STOP:
		IF fbSequenceManager.getState() <> E_SequenceState.STOP THEN
			fbSequenceManager.stopSequence();
			stInputs.stSequenceManager.Sequence_Command := E_SequenceState.WAIT;
		END_IF
	E_SequenceState.HOLD:
		IF fbSequenceManager.getState() <> E_SequenceState.HOLD THEN
			fbSequenceManager.pauseSequence();
			stInputs.stSequenceManager.Sequence_Command := E_SequenceState.WAIT;
		END_IF
END_CASE

(*
(*
			POP ACTUATORS
*)

fbLinAct_POP1.setMode(Mode := stInputs.stLinAct_POP1.Mode);
IF fbLinAct_POP1.inManual() THEN
	fbLinAct_POP1.setCommand(StateTarget := stInputs.stLinAct_POP1.Command);
ELSE
	stInputs.stLinAct_POP1.Command := fbLinAct_POP1.getCommand();
END_IF


fbLinAct_POP2.setMode(Mode := stInputs.stLinAct_POP2.Mode);
IF fbLinAct_POP2.inManual() THEN
	fbLinAct_POP2.setCommand(StateTarget := stInputs.stLinAct_POP2.Command);
ELSE
	stInputs.stLinAct_POP2.Command := fbLinAct_POP2.getCommand();
END_IF

fbLinAct_POP3.setMode(Mode := stInputs.stLinAct_POP3.Mode);
IF fbLinAct_POP3.inManual() THEN
	fbLinAct_POP3.setCommand(StateTarget := stInputs.stLinAct_POP3.Command);
ELSE
	stInputs.stLinAct_POP3.Command := fbLinAct_POP3.getCommand();
END_IF


(*
			TRAY CENTRE ACTUATORS
*)

fbTrayCentre_POP1.setMode(Mode := stInputs.stTrayCentre_POP1.Mode);
IF fbTrayCentre_POP1.inManual() THEN
	fbTrayCentre_POP1.setCommand(StateTarget := stInputs.stTrayCentre_POP1.Command);
ELSE
	stInputs.stTrayCentre_POP1.Command := fbTrayCentre_POP1.getCommand();
END_IF

fbTrayCentre_POP2.setMode(Mode := stInputs.stTrayCentre_POP2.Mode);
IF fbTrayCentre_POP2.inManual() THEN
	fbTrayCentre_POP2.setCommand(StateTarget := stInputs.stTrayCentre_POP2.Command);
ELSE
	stInputs.stTrayCentre_POP2.Command := fbTrayCentre_POP2.getCommand();
END_IF

fbTrayCentre_POP3.setMode(Mode := stInputs.stTrayCentre_POP3.Mode);
IF fbTrayCentre_POP3.inManual() THEN
	fbTrayCentre_POP3.setCommand(StateTarget := stInputs.stTrayCentre_POP3.Command);
ELSE
	stInputs.stTrayCentre_POP3.Command := fbTrayCentre_POP3.getCommand();
END_IF



(*
			STATIC CONVEYORS
*)


fbStaticConv_POP1.setMode(Mode := stInputs.stStaticConv_POP1.Mode);
IF fbStaticConv_POP1.inManual() THEN
	fbStaticConv_POP1.setCommand(StateTarget := stInputs.stStaticConv_POP1.Command);
ELSE
	stInputs.stStaticConv_POP1.Command := fbStaticConv_POP1.getCommand();
END_IF
									
fbStaticConv_POP2.setMode(Mode := stInputs.stStaticConv_POP2.Mode);
IF fbStaticConv_POP2.inManual() THEN
	fbStaticConv_POP2.setCommand(StateTarget := stInputs.stStaticConv_POP2.Command);
ELSE
	stInputs.stStaticConv_POP2.Command := fbStaticConv_POP2.getCommand();
END_IF

fbStaticConv_POP3.setMode(Mode := stInputs.stStaticConv_POP3.Mode);
IF fbStaticConv_POP3.inManual() THEN
	fbStaticConv_POP3.setCommand(StateTarget := stInputs.stStaticConv_POP3.Command);
ELSE
	stInputs.stStaticConv_POP3.Command := fbStaticConv_POP3.getCommand();
END_IF													


*)
END_METHOD

METHOD sequence : BOOL
VAR_INPUT
END_VAR
(*

IF (fbSequenceManager.getState() = E_SequenceState.COMPLETE) AND (fbHandshakeUpstream.stTrayExchgangeOutput.eState = E_TrayExchangeState.REQUESTED) AND NOT bInProgress THEN
	
	CASE ePOP_Type OF 
		E_POP_Type.EXTEND_CONVEY:
			fbSequenceManager.selectSequence(Sequence := E_SequenceList_POP.SEQ_EXTEND_CONVEY);
		E_POP_Type.CONVEY_EXTEND:
			fbSequenceManager.selectSequence(Sequence := E_SequenceList_POP.SEQ_CONVEY_EXTEND);
		E_POP_Type.RETRACT_CONVEY:
			fbSequenceManager.selectSequence(Sequence := E_SequenceList_POP.SEQ_RETRACT_CONVEY);
		E_POP_Type.CONVEY_RETRACT:
			fbSequenceManager.selectSequence(Sequence := E_SequenceList_POP.SEQ_RETRACT_CONVEY);
	END_CASE

	fbSequenceManager.startSequence();
	bInProgress := TRUE;
END_IF



IF (fbSequenceManager.getState() = E_SequenceState.COMPLETE) AND bInProgress THEN
	// return the pop conveyor back to resting condition
	CASE ePOP_Type OF 
		E_POP_Type.EXTEND_CONVEY:
			fbSequenceManager.selectSequence(Sequence := E_SequenceList_POP.SEQ_RETRACT);
		E_POP_Type.CONVEY_EXTEND:
			fbSequenceManager.selectSequence(Sequence := E_SequenceList_POP.SEQ_RETRACT);
		E_POP_Type.RETRACT_CONVEY:
			fbSequenceManager.selectSequence(Sequence := E_SequenceList_POP.SEQ_EXTEND);
		E_POP_Type.CONVEY_RETRACT:
			fbSequenceManager.selectSequence(Sequence := E_SequenceList_POP.SEQ_EXTEND);
	END_CASE
	fbSequenceManager.startSequence();
	bInProgress := FALSE;
END_IF

*)
END_METHOD

METHOD sequence_init : BOOL
VAR_INPUT
END_VAR
(*fbSeq_MOVE(devices := stAllComponents, bExt_1_Ret_0_Step2 := bExt_Step2, bExt_1_Ret_0_Step8 := bExt_Step8);
fbSeq_MOVE.populateSteps();
aSeqs[1] := fbSeq_MOVE;
*)
(*
fbSeq_RET_CONV(devices := stAllComponents);
fbSeq_CONV_EXT(devices := stAllComponents);
fbSeq_CONV_RET(devices := stAllComponents);
fbSeq_EXT(devices := stAllComponents);
fbSeq_RET(devices := stAllComponents);
*)


(*
fbSeqRND_DMMain(devices := stAllComponents);
fbSeqRND_DMCal(devices := stAllComponents);
fbSeqRND_DMFill(devices := stAllComponents);
fbSeqRND_DMDrain(devices := stAllComponents);
fbSeqRND_DMFlush(devices := stAllComponents);

fbSeqRND_DMMain.populateSteps();
fbSeqRND_DMCal.populateSteps();
fbSeqRND_DMFill.populateSteps();
fbSeqRND_DMDrain.populateSteps();
fbSeqRND_DMFlush.populateSteps();

aSeqs[1] := fbSeqRND_DMMain;
aSeqs[2] := fbSeqRND_DMCal;
aSeqs[3] := fbSeqRND_DMFill;
aSeqs[4] := fbSeqRND_DMDrain;
aSeqs[5] := fbSeqRND_DMFlush;


*)
END_METHOD

END_FUNCTION_BLOCK

// ---- POUs/00 Interfaces/FB_BaseMachine.TcPOU
{attribute 'OPC.UA.DA.StructuredType' := '1'}
FUNCTION_BLOCK FB_BaseMachine
VAR

	{attribute 'OPC.UA.DA' := '0'} 
	bBusy: BOOL := FALSE;
	{attribute 'OPC.UA.DA' := '1'} 
	bError: BOOL := FALSE;
	{attribute 'OPC.UA.DA' := '1'} 
	bEnable: BOOL := FALSE;
	{attribute 'OPC.UA.DA' := '1'} 
	eState: E_MachineState := E_MachineState.IDLE;
	{attribute 'OPC.UA.DA' := '1'} 
	{attribute 'OPC.UA.DA.StructuredType' := '1'}
	fbSequenceManager: FB_SequenceManager;
	{attribute 'OPC.UA.DA' := '0'} 
	aAllComponents: ARRAY[1..50] OF POINTER TO FB_BaseDevice;
	
	{attribute 'OPC.UA.DA' := '1'} 
	aErrors: ARRAY[1..20] OF ST_Alarm;	// raiseEvent() method updates Error1 / aErrors[1] only at the moment, must implement a ring buffer with error active checking for full functionality

	
END_VAR 

VAR_INPUT
	{attribute 'OPC.UA.DA' := '1'} 
	sID: STRING;  
	{attribute 'OPC.UA.DA' := '1'} 
	sDescr: STRING;
	{attribute 'OPC.UA.DA' := '1'} 
	nQtyComponents: INT;
END_VAR

METHOD devices_disable_All : BOOL
VAR
	iterator: INT;
	
END_VAR
FOR iterator:=1 TO nQtyComponents BY 1 DO
	aAllComponents[iterator]^.disable();
END_FOR
END_METHOD

METHOD devices_disable_CurrSeq : BOOL
VAR
	iterator: INT;
	Steps : ARRAY[1..20] OF ST_SequenceStep;
END_VAR
FOR iterator:=1 TO fbSequenceManager.getCurrentSeq_FB()^.stepsTotal() BY 1 DO
	
	Steps := fbSequenceManager.getCurrentSeq_FB()^.steps();
	Steps[iterator].Device^.disable();
	
END_FOR
END_METHOD

METHOD devices_enable_All : BOOL
VAR
	iterator: INT;
END_VAR
FOR iterator:=1 TO nQtyComponents BY 1 DO
	aAllComponents[iterator]^.enable();
END_FOR
END_METHOD

METHOD devices_enable_CurrSeq : BOOL
VAR
	iterator: INT;
	Steps : ARRAY[1..20] OF ST_SequenceStep;
END_VAR
FOR iterator:=1 TO fbSequenceManager.getCurrentSeq_FB()^.stepsTotal() BY 1 DO
	Steps := fbSequenceManager.getCurrentSeq_FB()^.steps();
	Steps[iterator].Device^.enable();
END_FOR
END_METHOD

METHOD devices_setAuto_All : BOOL
VAR
	iterator: INT;
END_VAR
FOR iterator:=1 TO nQtyComponents BY 1 DO
	aAllComponents[iterator]^.setMode(Mode := E_DeviceMode.AUTO);
END_FOR
END_METHOD

METHOD devices_setAuto_CurrSeq : BOOL
VAR
	iterator: INT;
	Steps : ARRAY[1..20] OF ST_SequenceStep;
END_VAR
FOR iterator:=1 TO fbSequenceManager.getCurrentSeq_FB()^.stepsTotal() BY 1 DO
	
	Steps := fbSequenceManager.getCurrentSeq_FB()^.steps();
	Steps[iterator].Device^.setMode(Mode := E_DeviceMode.AUTO);
END_FOR
END_METHOD

METHOD devices_setManual_All : BOOL
VAR
	iterator: INT;
END_VAR
FOR iterator:=1 TO nQtyComponents BY 1 DO
	aAllComponents[iterator]^.setMode(Mode := E_DeviceMode.AUTO);
END_FOR
END_METHOD

METHOD devices_setManual_CurrSeq : BOOL
VAR
	iterator: INT;
	Steps : ARRAY[1..20] OF ST_SequenceStep;
END_VAR
FOR iterator:=1 TO fbSequenceManager.getCurrentSeq_FB()^.stepsTotal() BY 1 DO
	
	Steps := fbSequenceManager.getCurrentSeq_FB()^.steps();
	Steps[iterator].Device^.setMode(Mode := E_DeviceMode.MANUAL);
END_FOR
END_METHOD

METHOD seq_Pause : BOOL
VAR_INPUT
END_VAR
fbSequenceManager.pauseSequence();
END_METHOD

METHOD seq_Start : BOOL
VAR_INPUT
	SeqNum: UINT;
END_VAR
devices_disable_All();
fbSequenceManager.selectSequence(Sequence := 1);
devices_enable_CurrSeq();
fbSequenceManager.startSequence();
END_METHOD

METHOD seq_Stop : BOOL
VAR_INPUT
END_VAR
fbSequenceManager.stopSequence();
END_METHOD

END_FUNCTION_BLOCK

// ---- POUs/05 Sequences/FB_SequenceManager.TcPOU
(*
		The sequence manager co-ordinates the selection and execution of 
		machine sequences. Machine sequences are created by extending the 
		FB_SequenceBase FB.
*)

FUNCTION_BLOCK FB_SequenceManager
VAR	
	//aSequences: ARRAY[1..5] OF POINTER TO FB_SequenceBase;
	 
	nNumberSequences: INT := 0;
	
	{attribute 'OPC.UA.DA' := '1'} 
	eState:  E_SequenceState := E_SequenceState.STOP; //always stop sequences after PLC restart
	{attribute 'OPC.UA.DA' := '1'} 
	eStateTarget:  E_SequenceState := E_SequenceState.STOP;
	
	eSMState: (STOPPED, STARTING, RUNNING, HOLD, COMPLETE) := STOPPED;
	nCurrentStep: INT := 1;
	nCurrentStepPreviousCycle: INT := 1;
	nCurrentSequence: INT := 1;
	nCurrentStepCheck: INT := 1; // use this to iterate over the sequence steps to check if an interlock has rolled back the sequence
	bPauseAcknowledged: BOOL := FALSE;
	
	{attribute 'OPC.UA.DA' := '0'} 
	fbTONstep: TON;			// these timers are set using the time values stored in each ST_SequenceStep
	{attribute 'OPC.UA.DA' := '0'} 
	fbTONdelay: TON;
	{attribute 'OPC.UA.DA' := '0'} 
	bIsFirstRun: BOOL := TRUE;
	
	i: INT;
	Steps : ARRAY[1..20] OF ST_SequenceStep;
	
	fbCurrentSequence: FB_SequenceBase;
END_VAR

VAR_IN_OUT
	aSequences: ARRAY[1..10] OF FB_SequenceBase;
	//fbCurrentSequence: FB_SequenceBase;
END_VAR

IF bIsFirstRun THEN
	fbTONdelay.PT := T#0S;
	fbTONdelay.IN := TRUE;
	fbTONdelay.PT := T#0S;
	fbTONstep.IN := FALSE;
	bIsFirstRun := FALSE;
	fbCurrentSequence := aSequences[1];
	eSMState := STOPPED;
END_IF

fbTONstep();
fbTONdelay();

CASE eSMState OF
	
	STOPPED:
		// Wait here until a start sequence command is received
		eState := E_SequenceState.STOP;
		
